   1:L PR[91] R[100]mm/sec CNT100;
   1:  PR[GP1:91,1] = PR[GP1:90,1] + 8.186;
   1:  PR[GP1:91,2] = PR[GP1:90,2] + 28.970;
   1:L PR[91] R[100]mm/sec CNT100;
   1:  PR[GP1:91,1] = PR[GP1:90,1] + 5.674;
   1:  PR[GP1:91,2] = PR[GP1:90,2] + 27.004;
   1:L PR[91] R[100]mm/sec CNT100;
   1:  PR[GP1:91,1] = PR[GP1:90,1] + 3.715;
   1:  PR[GP1:91,2] = PR[GP1:90,2] + 24.724;
   1:L PR[91] R[100]mm/sec CNT100;
   1:  PR[GP1:91,1] = PR[GP1:90,1] + 2.513;
   1:  PR[GP1:91,2] = PR[GP1:90,2] + 24.250;
   1:L PR[91] R[100]mm/sec CNT100;
   1:  PR[GP1:91,1] = PR[GP1:90,1] + 0.919;
   1:  PR[GP1:91,2] = PR[GP1:90,2] + 23.435;
   1:L PR[91] R[100]mm/sec CNT100;
   1:  ! -- Layer/Ebene 80 -- !;
   1:  PR[91] = PR[90];
   1:  PR[GP1:91,1] = PR[GP1:90,1] + -1.655;
   1:  PR[GP1:91,2] = PR[GP1:90,2] + 24.101;
   1:  PR[GP1:91,3] = PR[GP1:90,3] + 49.105;
   1:L PR[91] R[100]mm/sec CNT100;
   1:  PR[GP1:91,1] = PR[GP1:90,1] + -3.489;
   1:  PR[GP1:91,2] = PR[GP1:90,2] + 25.034;
   1:L PR[91] R[100]mm/sec CNT100;
   1:  PR[GP1:91,1] = PR[GP1:90,1] + -5.284;
   1:  PR[GP1:91,2] = PR[GP1:90,2] + 27.120;
   1:L PR[91] R[100]mm/sec CNT100;
   1:  PR[GP1:91,1] = PR[GP1:90,1] + -7.635;
   1:  PR[GP1:91,2] = PR[GP1:90,2] + 28.962;
   1:L PR[91] R[100]mm/sec CNT100;
   1:  PR[GP1:91,1] = PR[GP1:90,1] + -9.445;
   1:  PR[GP1:91,2] = PR[GP1:90,2] + 30.241;
   1:L PR[91] R[100]mm/sec CNT100;
   1:  PR[GP1:91,1] = PR[GP1:90,1] + -13.693;
   1:  PR[GP1:91,2] = PR[GP1:90,2] + 32.463;
   1:L PR[91] R[100]mm/sec CNT100;
   1:  PR[GP1:91,1] = PR[GP1:90,1] + -18.902;
   1:  PR[GP1:91,2] = PR[GP1:90,2] + 34.137;
   1:L PR[91] R[100]mm/sec CNT100;
   1:  PR[GP1:91,1] = PR[GP1:90,1] + -22.012;
   1:  PR[GP1:91,2] = PR[GP1:90,2] + 35.212;
   1:L PR[91] R[100]mm/sec CNT100;
   1:  PR[GP1:91,1] = PR[GP1:90,1] + -27.561;
   1:  PR[GP1:91,2] = PR[GP1:90,2] + 35.937;
   1:L PR[91] R[100]mm/sec CNT100;
   1:  PR[GP1:91,1] = PR[GP1:90,1] + -34.042;
   1:  PR[GP1:91,2] = PR[GP1:90,2] + 35.714;
   1:L PR[91] R[100]mm/sec CNT100;
   1:  PR[GP1:91,1] = PR[GP1:90,1] + -35.623;
   1:  PR[GP1:91,2] = PR[GP1:90,2] + 35.706;
   1:L PR[91] R[100]mm/sec CNT100;
   1:  PR[GP1:91,1] = PR[GP1:90,1] + -41.958;
   1:  PR[GP1:91,2] = PR[GP1:90,2] + 34.340;
   1:L PR[91] R[100]mm/sec CNT100;
   1:  PR[GP1:91,1] = PR[GP1:90,1] + -48.493;
   1:  PR[GP1:91,2] = PR[GP1:90,2] + 31.756;
   1:L PR[91] R[100]mm/sec CNT100;
   1:  PR[GP1:91,1] = PR[GP1:90,1] + -48.846;
   1:  PR[GP1:91,2] = PR[GP1:90,2] + 31.555;
   1:L PR[91] R[100]mm/sec CNT100;
   1:  PR[GP1:91,1] = PR[GP1:90,1] + -54.466;
   1:  PR[GP1:91,2] = PR[GP1:90,2] + 28.074;
   1:L PR[91] R[100]mm/sec CNT100;
   1:  PR[GP1:91,1] = PR[GP1:90,1] + -58.125;
   1:  PR[GP1:91,2] = PR[GP1:90,2] + 24.793;
   1:L PR[91] R[100]mm/sec CNT100;
   1:  PR[GP1:91,1] = PR[GP1:90,1] + -60.260;
   1:  PR[GP1:91,2] = PR[GP1:90,2] + 22.549;
   1:L PR[91] R[100]mm/sec CNT100;
   1:  PR[GP1:91,1] = PR[GP1:90,1] + -62.974;
   1:  PR[GP1:91,2] = PR[GP1:90,2] + 19.027;
   1:L PR[91] R[100]mm/sec CNT100;
   1:  PR[GP1:91,1] = PR[GP1:90,1] + -66.753;
   1:  PR[GP1:91,2] = PR[GP1:90,2] + 11.501;
   1:L PR[91] R[100]mm/sec CNT100;
   1:  PR[GP1:91,1] = PR[GP1:90,1] + -67.720;
   1:  PR[GP1:91,2] = PR[GP1:90,2] + 8.218;
   1:L PR[91] R[100]mm/sec CNT100;
   1:  PR[GP1:91,1] = PR[GP1:90,1] + -68.513;
   1:  PR[GP1:91,2] = PR[GP1:90,2] + 3.130;
   1:L PR[91] R[100]mm/sec CNT100;
   1:  PR[GP1:91,1] = PR[GP1:90,1] + -68.799;
   1:  PR[GP1:91,2] = PR[GP1:90,2] + -0.052;
   1:L PR[91] R[100]mm/sec CNT100;
   1:  PR[GP1:91,1] = PR[GP1:90,1] + -68.008;
   1:  PR[GP1:91,2] = PR[GP1:90,2] + -5.062;
   1:L PR[91] R[100]mm/sec CNT100;
   1:  PR[GP1:91,1] = PR[GP1:90,1] + -67.714;
   1:  PR[GP1:91,2] = PR[GP1:90,2] + -8.382;
   1:L PR[91] R[100]mm/sec CNT100;
   1:  PR[GP1:91,1] = PR[GP1:90,1] + -66.753;
   1:  PR[GP1:91,2] = PR[GP1:90,2] + -11.645;
   1:L PR[91] R[100]mm/sec CNT100;
   1:  PR[GP1:91,1] = PR[GP1:90,1] + -62.974;
   1:  PR[GP1:91,2] = PR[GP1:90,2] + -19.171;
   1:L PR[91] R[100]mm/sec CNT100;
   1:  PR[GP1:91,1] = PR[GP1:90,1] + -60.260;
   1:  PR[GP1:91,2] = PR[GP1:90,2] + -22.693;
   1:L PR[91] R[100]mm/sec CNT100;
   1:  PR[GP1:91,1] = PR[GP1:90,1] + -58.125;
   1:  PR[GP1:91,2] = PR[GP1:90,2] + -24.937;
   1:L PR[91] R[100]mm/sec CNT100;
   1:  PR[GP1:91,1] = PR[GP1:90,1] + -54.475;
   1:  PR[GP1:91,2] = PR[GP1:90,2] + -28.209;
   1:L PR[91] R[100]mm/sec CNT100;
   1:  PR[GP1:91,1] = PR[GP1:90,1] + -53.023;
   1:  PR[GP1:91,2] = PR[GP1:90,2] + -29.026;
   1:L PR[91] R[100]mm/sec CNT100;
   1:  PR[GP1:91,1] = PR[GP1:90,1] + -48.478;
   1:  PR[GP1:91,2] = PR[GP1:90,2] + -31.906;
   1:L PR[91] R[100]mm/sec CNT100;
   1:  PR[GP1:91,1] = PR[GP1:90,1] + -42.525;
   1:  PR[GP1:91,2] = PR[GP1:90,2] + -34.285;
   1:L PR[91] R[100]mm/sec CNT100;
   1:  PR[GP1:91,1] = PR[GP1:90,1] + -41.968;
   1:  PR[GP1:91,2] = PR[GP1:90,2] + -34.481;
   1:L PR[91] R[100]mm/sec CNT100;
   1:  PR[GP1:91,1] = PR[GP1:90,1] + -35.611;
   1:  PR[GP1:91,2] = PR[GP1:90,2] + -35.853;
   1:L PR[91] R[100]mm/sec CNT100;
   1:  PR[GP1:91,1] = PR[GP1:90,1] + -29.859;
   1:  PR[GP1:91,2] = PR[GP1:90,2] + -36.074;
   1:L PR[91] R[100]mm/sec CNT100;
   1:  PR[GP1:91,1] = PR[GP1:90,1] + -27.566;
   1:  PR[GP1:91,2] = PR[GP1:90,2] + -36.082;
   1:L PR[91] R[100]mm/sec CNT100;
   1:  PR[GP1:91,1] = PR[GP1:90,1] + -22.000;
   1:  PR[GP1:91,2] = PR[GP1:90,2] + -35.354;
   1:L PR[91] R[100]mm/sec CNT100;
   1:  PR[GP1:91,1] = PR[GP1:90,1] + -17.241;
   1:  PR[GP1:91,2] = PR[GP1:90,2] + -33.840;
   1:L PR[91] R[100]mm/sec CNT100;
   1:  PR[GP1:91,1] = PR[GP1:90,1] + -13.693;
   1:  PR[GP1:91,2] = PR[GP1:90,2] + -32.607;
   1:L PR[91] R[100]mm/sec CNT100;
   1:  PR[GP1:91,1] = PR[GP1:90,1] + -9.445;
   1:  PR[GP1:91,2] = PR[GP1:90,2] + -30.384;
   1:L PR[91] R[100]mm/sec CNT100;
   1:  PR[GP1:91,1] = PR[GP1:90,1] + -6.941;
   1:  PR[GP1:91,2] = PR[GP1:90,2] + -28.565;
   1:L PR[91] R[100]mm/sec CNT100;
   1:  PR[GP1:91,1] = PR[GP1:90,1] + -4.974;
   1:  PR[GP1:91,2] = PR[GP1:90,2] + -27.025;
   1:L PR[91] R[100]mm/sec CNT100;
   1:  PR[GP1:91,1] = PR[GP1:90,1] + -3.432;
   1:  PR[GP1:91,2] = PR[GP1:90,2] + -25.237;
   1:L PR[91] R[100]mm/sec CNT100;
   1:  PR[GP1:91,1] = PR[GP1:90,1] + -0.633;
   1:  PR[GP1:91,2] = PR[GP1:90,2] + -24.636;
   1:L PR[91] R[100]mm/sec CNT100;
   1:  PR[GP1:91,1] = PR[GP1:90,1] + 0.846;
   1:  PR[GP1:91,2] = PR[GP1:90,2] + -23.852;
   1:L PR[91] R[100]mm/sec CNT100;
   1:  PR[GP1:91,1] = PR[GP1:90,1] + 3.702;
   1:  PR[GP1:91,2] = PR[GP1:90,2] + -25.300;
   1:L PR[91] R[100]mm/sec CNT100;
   1:  PR[GP1:91,1] = PR[GP1:90,1] + 5.203;
   1:  PR[GP1:91,2] = PR[GP1:90,2] + -27.043;
   1:L PR[91] R[100]mm/sec CNT100;
   1:  PR[GP1:91,1] = PR[GP1:90,1] + 7.161;
   1:  PR[GP1:91,2] = PR[GP1:90,2] + -28.575;
   1:L PR[91] R[100]mm/sec CNT100;
   1:  PR[GP1:91,1] = PR[GP1:90,1] + 9.670;
   1:  PR[GP1:91,2] = PR[GP1:90,2] + -30.398;
   1:L PR[91] R[100]mm/sec CNT100;
   1:  PR[GP1:91,1] = PR[GP1:90,1] + 13.886;
   1:  PR[GP1:91,2] = PR[GP1:90,2] + -32.598;
   1:L PR[91] R[100]mm/sec CNT100;
   1:  PR[GP1:91,1] = PR[GP1:90,1] + 19.101;
   1:  PR[GP1:91,2] = PR[GP1:90,2] + -34.273;
   1:L PR[91] R[100]mm/sec CNT100;
   1:  PR[GP1:91,1] = PR[GP1:90,1] + 22.216;
   1:  PR[GP1:91,2] = PR[GP1:90,2] + -35.352;
   1:L PR[91] R[100]mm/sec CNT100;
   1:  PR[GP1:91,1] = PR[GP1:90,1] + 27.757;
   1:  PR[GP1:91,2] = PR[GP1:90,2] + -36.080;
   1:L PR[91] R[100]mm/sec CNT100;
   1:  PR[GP1:91,1] = PR[GP1:90,1] + 34.208;
   1:  PR[GP1:91,2] = PR[GP1:90,2] + -35.863;
   1:L PR[91] R[100]mm/sec CNT100;
   1:  PR[GP1:91,1] = PR[GP1:90,1] + 35.795;
   1:  PR[GP1:91,2] = PR[GP1:90,2] + -35.856;
   1:L PR[91] R[100]mm/sec CNT100;
   1:  PR[GP1:91,1] = PR[GP1:90,1] + 42.121;
   1:  PR[GP1:91,2] = PR[GP1:90,2] + -34.495;
   1:L PR[91] R[100]mm/sec CNT100;
   1:  PR[GP1:91,1] = PR[GP1:90,1] + 48.675;
   1:  PR[GP1:91,2] = PR[GP1:90,2] + -31.916;
   1:L PR[91] R[100]mm/sec CNT100;
   1:  PR[GP1:91,1] = PR[GP1:90,1] + 49.019;
   1:  PR[GP1:91,2] = PR[GP1:90,2] + -31.721;
   1:L PR[91] R[100]mm/sec CNT100;
   1:  PR[GP1:91,1] = PR[GP1:90,1] + 54.625;
   1:  PR[GP1:91,2] = PR[GP1:90,2] + -28.264;
   1:L PR[91] R[100]mm/sec CNT100;
   1:  PR[GP1:91,1] = PR[GP1:90,1] + 58.282;
   1:  PR[GP1:91,2] = PR[GP1:90,2] + -24.997;
   1:L PR[91] R[100]mm/sec CNT100;
   1:  PR[GP1:91,1] = PR[GP1:90,1] + 60.409;
   1:  PR[GP1:91,2] = PR[GP1:90,2] + -22.753;
   1:L PR[91] R[100]mm/sec CNT100;
   1:  PR[GP1:91,1] = PR[GP1:90,1] + 63.163;
   1:  PR[GP1:91,2] = PR[GP1:90,2] + -19.189;
   1:L PR[91] R[100]mm/sec CNT100;
   1:  PR[GP1:91,1] = PR[GP1:90,1] + 65.072;
   1:  PR[GP1:91,2] = PR[GP1:90,2] + -15.389;
   1:L PR[91] R[100]mm/sec CNT100;
   1:  PR[GP1:91,1] = PR[GP1:90,1] + 66.952;
   1:  PR[GP1:91,2] = PR[GP1:90,2] + -11.706;
   1:L PR[91] R[100]mm/sec CNT100;
   1:  PR[GP1:91,1] = PR[GP1:90,1] + 67.918;
   1:  PR[GP1:91,2] = PR[GP1:90,2] + -8.468;
   1:L PR[91] R[100]mm/sec CNT100;
   1:  PR[GP1:91,1] = PR[GP1:90,1] + 68.711;
   1:  PR[GP1:91,2] = PR[GP1:90,2] + -3.366;
   1:L PR[91] R[100]mm/sec CNT100;
   1:  PR[GP1:91,1] = PR[GP1:90,1] + 69.012;
   1:  PR[GP1:91,2] = PR[GP1:90,2] + -0.092;
   1:L PR[91] R[100]mm/sec CNT100;
   1:  PR[GP1:91,1] = PR[GP1:90,1] + 68.221;
   1:  PR[GP1:91,2] = PR[GP1:90,2] + 4.931;
   1:L PR[91] R[100]mm/sec CNT100;
   1:  PR[GP1:91,1] = PR[GP1:90,1] + 67.912;
   1:  PR[GP1:91,2] = PR[GP1:90,2] + 8.343;
   1:L PR[91] R[100]mm/sec CNT100;
   1:  PR[GP1:91,1] = PR[GP1:90,1] + 66.951;
   1:  PR[GP1:91,2] = PR[GP1:90,2] + 11.564;
   1:L PR[91] R[100]mm/sec CNT100;
   1:  PR[GP1:91,1] = PR[GP1:90,1] + 64.946;
   1:  PR[GP1:91,2] = PR[GP1:90,2] + 15.559;
   1:L PR[91] R[100]mm/sec CNT100;
   1:  PR[GP1:91,1] = PR[GP1:90,1] + 63.164;
   1:  PR[GP1:91,2] = PR[GP1:90,2] + 19.044;
   1:L PR[91] R[100]mm/sec CNT100;
   1:  PR[GP1:91,1] = PR[GP1:90,1] + 60.409;
   1:  PR[GP1:91,2] = PR[GP1:90,2] + 22.609;
   1:L PR[91] R[100]mm/sec CNT100;
   1:  PR[GP1:91,1] = PR[GP1:90,1] + 58.282;
   1:  PR[GP1:91,2] = PR[GP1:90,2] + 24.853;
   1:L PR[91] R[100]mm/sec CNT100;
   1:  PR[GP1:91,1] = PR[GP1:90,1] + 54.634;
   1:  PR[GP1:91,2] = PR[GP1:90,2] + 28.112;
   1:L PR[91] R[100]mm/sec CNT100;
   1:  PR[GP1:91,1] = PR[GP1:90,1] + 53.192;
   1:  PR[GP1:91,2] = PR[GP1:90,2] + 28.923;
   1:L PR[91] R[100]mm/sec CNT100;
   1:  PR[GP1:91,1] = PR[GP1:90,1] + 48.661;
   1:  PR[GP1:91,2] = PR[GP1:90,2] + 31.778;
   1:L PR[91] R[100]mm/sec CNT100;
   1:  PR[GP1:91,1] = PR[GP1:90,1] + 42.696;
   1:  PR[GP1:91,2] = PR[GP1:90,2] + 34.150;
   1:L PR[91] R[100]mm/sec CNT100;
   1:  PR[GP1:91,1] = PR[GP1:90,1] + 42.133;
   1:  PR[GP1:91,2] = PR[GP1:90,2] + 34.349;
   1:L PR[91] R[100]mm/sec CNT100;
   1:  PR[GP1:91,1] = PR[GP1:90,1] + 35.787;
   1:  PR[GP1:91,2] = PR[GP1:90,2] + 35.714;
   1:L PR[91] R[100]mm/sec CNT100;
   1:  PR[GP1:91,1] = PR[GP1:90,1] + 30.063;
   1:  PR[GP1:91,2] = PR[GP1:90,2] + 35.930;
   1:L PR[91] R[100]mm/sec CNT100;
   1:  PR[GP1:91,1] = PR[GP1:90,1] + 27.770;
   1:  PR[GP1:91,2] = PR[GP1:90,2] + 35.938;
   1:L PR[91] R[100]mm/sec CNT100;
   1:  PR[GP1:91,1] = PR[GP1:90,1] + 22.213;
   1:  PR[GP1:91,2] = PR[GP1:90,2] + 35.208;
   1:L PR[91] R[100]mm/sec CNT100;
   1:  PR[GP1:91,1] = PR[GP1:90,1] + 17.448;
   1:  PR[GP1:91,2] = PR[GP1:90,2] + 33.692;
   1:L PR[91] R[100]mm/sec CNT100;
   1:  PR[GP1:91,1] = PR[GP1:90,1] + 13.898;
   1:  PR[GP1:91,2] = PR[GP1:90,2] + 32.461;
   1:L PR[91] R[100]mm/sec CNT100;
   1:  PR[GP1:91,1] = PR[GP1:90,1] + 9.670;
   1:  PR[GP1:91,2] = PR[GP1:90,2] + 30.255;
   1:L PR[91] R[100]mm/sec CNT100;
   1:  PR[GP1:91,1] = PR[GP1:90,1] + 7.856;
   1:  PR[GP1:91,2] = PR[GP1:90,2] + 28.973;
   1:L PR[91] R[100]mm/sec CNT100;
   1:  PR[GP1:91,1] = PR[GP1:90,1] + 5.516;
   1:  PR[GP1:91,2] = PR[GP1:90,2] + 27.142;
   1:L PR[91] R[100]mm/sec CNT100;
   1:  PR[GP1:91,1] = PR[GP1:90,1] + 3.685;
   1:  PR[GP1:91,2] = PR[GP1:90,2] + 25.011;
   1:L PR[91] R[100]mm/sec CNT100;
   1:  PR[GP1:91,1] = PR[GP1:90,1] + 2.424;
   1:  PR[GP1:91,2] = PR[GP1:90,2] + 24.513;
   1:L PR[91] R[100]mm/sec CNT100;
   1:  PR[GP1:91,1] = PR[GP1:90,1] + 0.960;
   1:  PR[GP1:91,2] = PR[GP1:90,2] + 23.765;
   1:L PR[91] R[100]mm/sec CNT100;
   1:  ! -- Layer/Ebene 81 -- !;
   1:  PR[91] = PR[90];
   1:  PR[GP1:91,1] = PR[GP1:90,1] + -1.744;
   1:  PR[GP1:91,2] = PR[GP1:90,2] + 24.447;
   1:  PR[GP1:91,3] = PR[GP1:90,3] + 49.715;
   1:L PR[91] R[100]mm/sec CNT100;
   1:  PR[GP1:91,1] = PR[GP1:90,1] + -3.460;
   1:  PR[GP1:91,2] = PR[GP1:90,2] + 25.320;
   1:L PR[91] R[100]mm/sec CNT100;
   1:  PR[GP1:91,1] = PR[GP1:90,1] + -5.128;
   1:  PR[GP1:91,2] = PR[GP1:90,2] + 27.260;
   1:L PR[91] R[100]mm/sec CNT100;
   1:  PR[GP1:91,1] = PR[GP1:90,1] + -7.305;
   1:  PR[GP1:91,2] = PR[GP1:90,2] + 28.965;
   1:L PR[91] R[100]mm/sec CNT100;
   1:  PR[GP1:91,1] = PR[GP1:90,1] + -9.235;
   1:  PR[GP1:91,2] = PR[GP1:90,2] + 30.328;
   1:L PR[91] R[100]mm/sec CNT100;
   1:  PR[GP1:91,1] = PR[GP1:90,1] + -13.351;
   1:  PR[GP1:91,2] = PR[GP1:90,2] + 32.482;
   1:L PR[91] R[100]mm/sec CNT100;
   1:  PR[GP1:91,1] = PR[GP1:90,1] + -18.401;
   1:  PR[GP1:91,2] = PR[GP1:90,2] + 34.104;
   1:L PR[91] R[100]mm/sec CNT100;
   1:  PR[GP1:91,1] = PR[GP1:90,1] + -21.813;
   1:  PR[GP1:91,2] = PR[GP1:90,2] + 35.284;
   1:L PR[91] R[100]mm/sec CNT100;
   1:  PR[GP1:91,1] = PR[GP1:90,1] + -27.209;
   1:  PR[GP1:91,2] = PR[GP1:90,2] + 35.989;
   1:L PR[91] R[100]mm/sec CNT100;
   1:  PR[GP1:91,1] = PR[GP1:90,1] + -33.514;
   1:  PR[GP1:91,2] = PR[GP1:90,2] + 35.773;
   1:L PR[91] R[100]mm/sec CNT100;
   1:  PR[GP1:91,1] = PR[GP1:90,1] + -35.435;
   1:  PR[GP1:91,2] = PR[GP1:90,2] + 35.763;
   1:L PR[91] R[100]mm/sec CNT100;
   1:  PR[GP1:91,1] = PR[GP1:90,1] + -41.613;
   1:  PR[GP1:91,2] = PR[GP1:90,2] + 34.430;
   1:L PR[91] R[100]mm/sec CNT100;
   1:  PR[GP1:91,1] = PR[GP1:90,1] + -48.418;
   1:  PR[GP1:91,2] = PR[GP1:90,2] + 31.741;
   1:L PR[91] R[100]mm/sec CNT100;
   1:  PR[GP1:91,1] = PR[GP1:90,1] + -54.253;
   1:  PR[GP1:91,2] = PR[GP1:90,2] + 28.124;
   1:L PR[91] R[100]mm/sec CNT100;
   1:  PR[GP1:91,1] = PR[GP1:90,1] + -58.181;
   1:  PR[GP1:91,2] = PR[GP1:90,2] + 24.602;
   1:L PR[91] R[100]mm/sec CNT100;
   1:  PR[GP1:91,1] = PR[GP1:90,1] + -59.893;
   1:  PR[GP1:91,2] = PR[GP1:90,2] + 22.802;
   1:L PR[91] R[100]mm/sec CNT100;
   1:  PR[GP1:91,1] = PR[GP1:90,1] + -62.849;
   1:  PR[GP1:91,2] = PR[GP1:90,2] + 18.966;
   1:L PR[91] R[100]mm/sec CNT100;
   1:  PR[GP1:91,1] = PR[GP1:90,1] + -66.536;
   1:  PR[GP1:91,2] = PR[GP1:90,2] + 11.628;
   1:L PR[91] R[100]mm/sec CNT100;
   1:  PR[GP1:91,1] = PR[GP1:90,1] + -67.603;
   1:  PR[GP1:91,2] = PR[GP1:90,2] + 8.004;
   1:L PR[91] R[100]mm/sec CNT100;
   1:  PR[GP1:91,1] = PR[GP1:90,1] + -68.306;
   1:  PR[GP1:91,2] = PR[GP1:90,2] + 3.493;
   1:L PR[91] R[100]mm/sec CNT100;
   1:  PR[GP1:91,1] = PR[GP1:90,1] + -68.625;
   1:  PR[GP1:91,2] = PR[GP1:90,2] + -0.052;
   1:L PR[91] R[100]mm/sec CNT100;
   1:  PR[GP1:91,1] = PR[GP1:90,1] + -67.921;
   1:  PR[GP1:91,2] = PR[GP1:90,2] + -4.508;
   1:L PR[91] R[100]mm/sec CNT100;
   1:  PR[GP1:91,1] = PR[GP1:90,1] + -67.597;
   1:  PR[GP1:91,2] = PR[GP1:90,2] + -8.168;
   1:L PR[91] R[100]mm/sec CNT100;
   1:  PR[GP1:91,1] = PR[GP1:90,1] + -66.536;
   1:  PR[GP1:91,2] = PR[GP1:90,2] + -11.772;
   1:L PR[91] R[100]mm/sec CNT100;
   1:  PR[GP1:91,1] = PR[GP1:90,1] + -62.849;
   1:  PR[GP1:91,2] = PR[GP1:90,2] + -19.110;
   1:L PR[91] R[100]mm/sec CNT100;
   1:  PR[GP1:91,1] = PR[GP1:90,1] + -59.893;
   1:  PR[GP1:91,2] = PR[GP1:90,2] + -22.946;
   1:L PR[91] R[100]mm/sec CNT100;
   1:  PR[GP1:91,1] = PR[GP1:90,1] + -58.181;
   1:  PR[GP1:91,2] = PR[GP1:90,2] + -24.746;
   1:L PR[91] R[100]mm/sec CNT100;
   1:  PR[GP1:91,1] = PR[GP1:90,1] + -54.262;
   1:  PR[GP1:91,2] = PR[GP1:90,2] + -28.259;
   1:L PR[91] R[100]mm/sec CNT100;
   1:  PR[GP1:91,1] = PR[GP1:90,1] + -53.300;
   1:  PR[GP1:91,2] = PR[GP1:90,2] + -28.801;
   1:L PR[91] R[100]mm/sec CNT100;
   1:  PR[GP1:91,1] = PR[GP1:90,1] + -48.414;
   1:  PR[GP1:91,2] = PR[GP1:90,2] + -31.887;
   1:L PR[91] R[100]mm/sec CNT100;
   1:  PR[GP1:91,1] = PR[GP1:90,1] + -42.479;
   1:  PR[GP1:91,2] = PR[GP1:90,2] + -34.270;
   1:L PR[91] R[100]mm/sec CNT100;
   1:  PR[GP1:91,1] = PR[GP1:90,1] + -41.622;
   1:  PR[GP1:91,2] = PR[GP1:90,2] + -34.572;
   1:L PR[91] R[100]mm/sec CNT100;
   1:  PR[GP1:91,1] = PR[GP1:90,1] + -35.423;
   1:  PR[GP1:91,2] = PR[GP1:90,2] + -35.909;
   1:L PR[91] R[100]mm/sec CNT100;
   1:  PR[GP1:91,1] = PR[GP1:90,1] + -29.813;
   1:  PR[GP1:91,2] = PR[GP1:90,2] + -36.126;
   1:L PR[91] R[100]mm/sec CNT100;
   1:  PR[GP1:91,1] = PR[GP1:90,1] + -27.214;
   1:  PR[GP1:91,2] = PR[GP1:90,2] + -36.134;
   1:L PR[91] R[100]mm/sec CNT100;
   1:  PR[GP1:91,1] = PR[GP1:90,1] + -21.801;
   1:  PR[GP1:91,2] = PR[GP1:90,2] + -35.426;
   1:L PR[91] R[100]mm/sec CNT100;
   1:  PR[GP1:91,1] = PR[GP1:90,1] + -17.172;
   1:  PR[GP1:91,2] = PR[GP1:90,2] + -33.953;
   1:L PR[91] R[100]mm/sec CNT100;
   1:  PR[GP1:91,1] = PR[GP1:90,1] + -13.351;
   1:  PR[GP1:91,2] = PR[GP1:90,2] + -32.625;
   1:L PR[91] R[100]mm/sec CNT100;
   1:  PR[GP1:91,1] = PR[GP1:90,1] + -9.234;
   1:  PR[GP1:91,2] = PR[GP1:90,2] + -30.472;
   1:L PR[91] R[100]mm/sec CNT100;
   1:  PR[GP1:91,1] = PR[GP1:90,1] + -6.567;
   1:  PR[GP1:91,2] = PR[GP1:90,2] + -28.534;
   1:L PR[91] R[100]mm/sec CNT100;
   1:  PR[GP1:91,1] = PR[GP1:90,1] + -4.801;
   1:  PR[GP1:91,2] = PR[GP1:90,2] + -27.151;
   1:L PR[91] R[100]mm/sec CNT100;
   1:  PR[GP1:91,1] = PR[GP1:90,1] + -3.403;
   1:  PR[GP1:91,2] = PR[GP1:90,2] + -25.530;
   1:L PR[91] R[100]mm/sec CNT100;
   1:  PR[GP1:91,1] = PR[GP1:90,1] + -0.466;
   1:  PR[GP1:91,2] = PR[GP1:90,2] + -24.899;
   1:L PR[91] R[100]mm/sec CNT100;
   1:  PR[GP1:91,1] = PR[GP1:90,1] + 0.887;
   1:  PR[GP1:91,2] = PR[GP1:90,2] + -24.182;
   1:L PR[91] R[100]mm/sec CNT100;
   1:  PR[GP1:91,1] = PR[GP1:90,1] + 3.672;
   1:  PR[GP1:91,2] = PR[GP1:90,2] + -25.593;
   1:L PR[91] R[100]mm/sec CNT100;
   1:  PR[GP1:91,1] = PR[GP1:90,1] + 5.028;
   1:  PR[GP1:91,2] = PR[GP1:90,2] + -27.168;
   1:L PR[91] R[100]mm/sec CNT100;
   1:  PR[GP1:91,1] = PR[GP1:90,1] + 6.786;
   1:  PR[GP1:91,2] = PR[GP1:90,2] + -28.543;
   1:L PR[91] R[100]mm/sec CNT100;
   1:  PR[GP1:91,1] = PR[GP1:90,1] + 9.459;
   1:  PR[GP1:91,2] = PR[GP1:90,2] + -30.485;
   1:L PR[91] R[100]mm/sec CNT100;
   1:  PR[GP1:91,1] = PR[GP1:90,1] + 13.544;
   1:  PR[GP1:91,2] = PR[GP1:90,2] + -32.617;
   1:L PR[91] R[100]mm/sec CNT100;
   1:  PR[GP1:91,1] = PR[GP1:90,1] + 18.599;
   1:  PR[GP1:91,2] = PR[GP1:90,2] + -34.241;
   1:L PR[91] R[100]mm/sec CNT100;
   1:  PR[GP1:91,1] = PR[GP1:90,1] + 22.017;
   1:  PR[GP1:91,2] = PR[GP1:90,2] + -35.424;
   1:L PR[91] R[100]mm/sec CNT100;
   1:  PR[GP1:91,1] = PR[GP1:90,1] + 27.405;
   1:  PR[GP1:91,2] = PR[GP1:90,2] + -36.133;
   1:L PR[91] R[100]mm/sec CNT100;
   1:  PR[GP1:91,1] = PR[GP1:90,1] + 33.681;
   1:  PR[GP1:91,2] = PR[GP1:90,2] + -35.921;
   1:L PR[91] R[100]mm/sec CNT100;
   1:  PR[GP1:91,1] = PR[GP1:90,1] + 35.608;
   1:  PR[GP1:91,2] = PR[GP1:90,2] + -35.913;
   1:L PR[91] R[100]mm/sec CNT100;
   1:  PR[GP1:91,1] = PR[GP1:90,1] + 41.777;
   1:  PR[GP1:91,2] = PR[GP1:90,2] + -34.585;
   1:L PR[91] R[100]mm/sec CNT100;
   1:  PR[GP1:91,1] = PR[GP1:90,1] + 48.597;
   1:  PR[GP1:91,2] = PR[GP1:90,2] + -31.903;
   1:L PR[91] R[100]mm/sec CNT100;
   1:  PR[GP1:91,1] = PR[GP1:90,1] + 54.408;
   1:  PR[GP1:91,2] = PR[GP1:90,2] + -28.317;
   1:L PR[91] R[100]mm/sec CNT100;
   1:  PR[GP1:91,1] = PR[GP1:90,1] + 58.334;
   1:  PR[GP1:91,2] = PR[GP1:90,2] + -24.809;
   1:L PR[91] R[100]mm/sec CNT100;
   1:  PR[GP1:91,1] = PR[GP1:90,1] + 60.037;
   1:  PR[GP1:91,2] = PR[GP1:90,2] + -23.013;
   1:L PR[91] R[100]mm/sec CNT100;
   1:  PR[GP1:91,1] = PR[GP1:90,1] + 63.036;
   1:  PR[GP1:91,2] = PR[GP1:90,2] + -19.131;
   1:L PR[91] R[100]mm/sec CNT100;
   1:  PR[GP1:91,1] = PR[GP1:90,1] + 64.662;
   1:  PR[GP1:91,2] = PR[GP1:90,2] + -15.896;
   1:L PR[91] R[100]mm/sec CNT100;
   1:  PR[GP1:91,1] = PR[GP1:90,1] + 66.733;
   1:  PR[GP1:91,2] = PR[GP1:90,2] + -11.836;
   1:L PR[91] R[100]mm/sec CNT100;
   1:  PR[GP1:91,1] = PR[GP1:90,1] + 67.800;
   1:  PR[GP1:91,2] = PR[GP1:90,2] + -8.262;
   1:L PR[91] R[100]mm/sec CNT100;
   1:  PR[GP1:91,1] = PR[GP1:90,1] + 68.503;
   1:  PR[GP1:91,2] = PR[GP1:90,2] + -3.740;
   1:L PR[91] R[100]mm/sec CNT100;
   1:  PR[GP1:91,1] = PR[GP1:90,1] + 68.838;
   1:  PR[GP1:91,2] = PR[GP1:90,2] + -0.092;
   1:L PR[91] R[100]mm/sec CNT100;
   1:  PR[GP1:91,1] = PR[GP1:90,1] + 68.134;
   1:  PR[GP1:91,2] = PR[GP1:90,2] + 4.377;
   1:L PR[91] R[100]mm/sec CNT100;
   1:  PR[GP1:91,1] = PR[GP1:90,1] + 67.794;
   1:  PR[GP1:91,2] = PR[GP1:90,2] + 8.137;
   1:L PR[91] R[100]mm/sec CNT100;
   1:  PR[GP1:91,1] = PR[GP1:90,1] + 66.733;
   1:  PR[GP1:91,2] = PR[GP1:90,2] + 11.694;
   1:L PR[91] R[100]mm/sec CNT100;
   1:  PR[GP1:91,1] = PR[GP1:90,1] + 64.977;
   1:  PR[GP1:91,2] = PR[GP1:90,2] + 15.191;
   1:L PR[91] R[100]mm/sec CNT100;
   1:  PR[GP1:91,1] = PR[GP1:90,1] + 63.037;
   1:  PR[GP1:91,2] = PR[GP1:90,2] + 18.986;
   1:L PR[91] R[100]mm/sec CNT100;
   1:  PR[GP1:91,1] = PR[GP1:90,1] + 60.037;
   1:  PR[GP1:91,2] = PR[GP1:90,2] + 22.869;
   1:L PR[91] R[100]mm/sec CNT100;
   1:  PR[GP1:91,1] = PR[GP1:90,1] + 58.334;
   1:  PR[GP1:91,2] = PR[GP1:90,2] + 24.665;
   1:L PR[91] R[100]mm/sec CNT100;
   1:  PR[GP1:91,1] = PR[GP1:90,1] + 54.417;
   1:  PR[GP1:91,2] = PR[GP1:90,2] + 28.165;
   1:L PR[91] R[100]mm/sec CNT100;
   1:  PR[GP1:91,1] = PR[GP1:90,1] + 53.466;
   1:  PR[GP1:91,2] = PR[GP1:90,2] + 28.700;
   1:L PR[91] R[100]mm/sec CNT100;
   1:  PR[GP1:91,1] = PR[GP1:90,1] + 48.593;
   1:  PR[GP1:91,2] = PR[GP1:90,2] + 31.761;
   1:L PR[91] R[100]mm/sec CNT100;
   1:  PR[GP1:91,1] = PR[GP1:90,1] + 42.650;
   1:  PR[GP1:91,2] = PR[GP1:90,2] + 34.135;
   1:L PR[91] R[100]mm/sec CNT100;
   1:  PR[GP1:91,1] = PR[GP1:90,1] + 41.788;
   1:  PR[GP1:91,2] = PR[GP1:90,2] + 34.439;
   1:L PR[91] R[100]mm/sec CNT100;
   1:  PR[GP1:91,1] = PR[GP1:90,1] + 35.600;
   1:  PR[GP1:91,2] = PR[GP1:90,2] + 35.771;
   1:L PR[91] R[100]mm/sec CNT100;
   1:  PR[GP1:91,1] = PR[GP1:90,1] + 30.018;
   1:  PR[GP1:91,2] = PR[GP1:90,2] + 35.981;
   1:L PR[91] R[100]mm/sec CNT100;
   1:  PR[GP1:91,1] = PR[GP1:90,1] + 27.419;
   1:  PR[GP1:91,2] = PR[GP1:90,2] + 35.990;
   1:L PR[91] R[100]mm/sec CNT100;
   1:  PR[GP1:91,1] = PR[GP1:90,1] + 22.014;
   1:  PR[GP1:91,2] = PR[GP1:90,2] + 35.280;
   1:L PR[91] R[100]mm/sec CNT100;
   1:  PR[GP1:91,1] = PR[GP1:90,1] + 17.380;
   1:  PR[GP1:91,2] = PR[GP1:90,2] + 33.805;
   1:L PR[91] R[100]mm/sec CNT100;
   1:  PR[GP1:91,1] = PR[GP1:90,1] + 13.556;
   1:  PR[GP1:91,2] = PR[GP1:90,2] + 32.480;
   1:L PR[91] R[100]mm/sec CNT100;
   1:  PR[GP1:91,1] = PR[GP1:90,1] + 9.459;
   1:  PR[GP1:91,2] = PR[GP1:90,2] + 30.341;
   1:L PR[91] R[100]mm/sec CNT100;
   1:  PR[GP1:91,1] = PR[GP1:90,1] + 7.525;
   1:  PR[GP1:91,2] = PR[GP1:90,2] + 28.975;
   1:L PR[91] R[100]mm/sec CNT100;
   1:  PR[GP1:91,1] = PR[GP1:90,1] + 5.358;
   1:  PR[GP1:91,2] = PR[GP1:90,2] + 27.280;
   1:L PR[91] R[100]mm/sec CNT100;
   1:  PR[GP1:91,1] = PR[GP1:90,1] + 3.655;
   1:  PR[GP1:91,2] = PR[GP1:90,2] + 25.298;
   1:L PR[91] R[100]mm/sec CNT100;
   1:  PR[GP1:91,1] = PR[GP1:90,1] + 2.335;
   1:  PR[GP1:91,2] = PR[GP1:90,2] + 24.776;
   1:L PR[91] R[100]mm/sec CNT100;
   1:  PR[GP1:91,1] = PR[GP1:90,1] + 1.001;
   1:  PR[GP1:91,2] = PR[GP1:90,2] + 24.095;
   1:L PR[91] R[100]mm/sec CNT100;
   1:  ! -- Layer/Ebene 82 -- !;
   1:  PR[91] = PR[90];
   1:  PR[GP1:91,1] = PR[GP1:90,1] + -1.832;
   1:  PR[GP1:91,2] = PR[GP1:90,2] + 24.794;
   1:  PR[GP1:91,3] = PR[GP1:90,3] + 50.325;
   1:L PR[91] R[100]mm/sec CNT100;
   1:  PR[GP1:91,1] = PR[GP1:90,1] + -3.430;
   1:  PR[GP1:91,2] = PR[GP1:90,2] + 25.607;
   1:L PR[91] R[100]mm/sec CNT100;
   1:  PR[GP1:91,1] = PR[GP1:90,1] + -4.972;
   1:  PR[GP1:91,2] = PR[GP1:90,2] + 27.399;
   1:L PR[91] R[100]mm/sec CNT100;
   1:  PR[GP1:91,1] = PR[GP1:90,1] + -6.976;
   1:  PR[GP1:91,2] = PR[GP1:90,2] + 28.969;
   1:L PR[91] R[100]mm/sec CNT100;
   1:  PR[GP1:91,1] = PR[GP1:90,1] + -9.024;
   1:  PR[GP1:91,2] = PR[GP1:90,2] + 30.416;
   1:L PR[91] R[100]mm/sec CNT100;
   1:  PR[GP1:91,1] = PR[GP1:90,1] + -13.009;
   1:  PR[GP1:91,2] = PR[GP1:90,2] + 32.501;
   1:L PR[91] R[100]mm/sec CNT100;
   1:  PR[GP1:91,1] = PR[GP1:90,1] + -17.900;
   1:  PR[GP1:91,2] = PR[GP1:90,2] + 34.072;
   1:L PR[91] R[100]mm/sec CNT100;
   1:  PR[GP1:91,1] = PR[GP1:90,1] + -21.615;
   1:  PR[GP1:91,2] = PR[GP1:90,2] + 35.356;
   1:L PR[91] R[100]mm/sec CNT100;
   1:  PR[GP1:91,1] = PR[GP1:90,1] + -26.858;
   1:  PR[GP1:91,2] = PR[GP1:90,2] + 36.042;
   1:L PR[91] R[100]mm/sec CNT100;
   1:  PR[GP1:91,1] = PR[GP1:90,1] + -32.986;
   1:  PR[GP1:91,2] = PR[GP1:90,2] + 35.831;
   1:L PR[91] R[100]mm/sec CNT100;
   1:  PR[GP1:91,1] = PR[GP1:90,1] + -35.247;
   1:  PR[GP1:91,2] = PR[GP1:90,2] + 35.820;
   1:L PR[91] R[100]mm/sec CNT100;
   1:  PR[GP1:91,1] = PR[GP1:90,1] + -41.267;
   1:  PR[GP1:91,2] = PR[GP1:90,2] + 34.521;
   1:L PR[91] R[100]mm/sec CNT100;
   1:  PR[GP1:91,1] = PR[GP1:90,1] + -47.841;
   1:  PR[GP1:91,2] = PR[GP1:90,2] + 31.918;
   1:L PR[91] R[100]mm/sec CNT100;
   1:  PR[GP1:91,1] = PR[GP1:90,1] + -48.243;
   1:  PR[GP1:91,2] = PR[GP1:90,2] + 31.775;
   1:L PR[91] R[100]mm/sec CNT100;
   1:  PR[GP1:91,1] = PR[GP1:90,1] + -54.039;
   1:  PR[GP1:91,2] = PR[GP1:90,2] + 28.174;
   1:L PR[91] R[100]mm/sec CNT100;
   1:  PR[GP1:91,1] = PR[GP1:90,1] + -58.237;
   1:  PR[GP1:91,2] = PR[GP1:90,2] + 24.411;
   1:L PR[91] R[100]mm/sec CNT100;
   1:  PR[GP1:91,1] = PR[GP1:90,1] + -59.526;
   1:  PR[GP1:91,2] = PR[GP1:90,2] + 23.055;
   1:L PR[91] R[100]mm/sec CNT100;
   1:  PR[GP1:91,1] = PR[GP1:90,1] + -62.724;
   1:  PR[GP1:91,2] = PR[GP1:90,2] + 18.904;
   1:L PR[91] R[100]mm/sec CNT100;
   1:  PR[GP1:91,1] = PR[GP1:90,1] + -66.320;
   1:  PR[GP1:91,2] = PR[GP1:90,2] + 11.754;
   1:L PR[91] R[100]mm/sec CNT100;
   1:  PR[GP1:91,1] = PR[GP1:90,1] + -67.486;
   1:  PR[GP1:91,2] = PR[GP1:90,2] + 7.790;
   1:L PR[91] R[100]mm/sec CNT100;
   1:  PR[GP1:91,1] = PR[GP1:90,1] + -68.100;
   1:  PR[GP1:91,2] = PR[GP1:90,2] + 3.857;
   1:L PR[91] R[100]mm/sec CNT100;
   1:  PR[GP1:91,1] = PR[GP1:90,1] + -68.451;
   1:  PR[GP1:91,2] = PR[GP1:90,2] + -0.052;
   1:L PR[91] R[100]mm/sec CNT100;
   1:  PR[GP1:91,1] = PR[GP1:90,1] + -67.834;
   1:  PR[GP1:91,2] = PR[GP1:90,2] + -3.955;
   1:L PR[91] R[100]mm/sec CNT100;
   1:  PR[GP1:91,1] = PR[GP1:90,1] + -67.481;
   1:  PR[GP1:91,2] = PR[GP1:90,2] + -7.953;
   1:L PR[91] R[100]mm/sec CNT100;
   1:  PR[GP1:91,1] = PR[GP1:90,1] + -66.320;
   1:  PR[GP1:91,2] = PR[GP1:90,2] + -11.898;
   1:L PR[91] R[100]mm/sec CNT100;
   1:  PR[GP1:91,1] = PR[GP1:90,1] + -62.724;
   1:  PR[GP1:91,2] = PR[GP1:90,2] + -19.048;
   1:L PR[91] R[100]mm/sec CNT100;
   1:  PR[GP1:91,1] = PR[GP1:90,1] + -59.526;
   1:  PR[GP1:91,2] = PR[GP1:90,2] + -23.199;
   1:L PR[91] R[100]mm/sec CNT100;
   1:  PR[GP1:91,1] = PR[GP1:90,1] + -58.237;
   1:  PR[GP1:91,2] = PR[GP1:90,2] + -24.555;
   1:L PR[91] R[100]mm/sec CNT100;
   1:  PR[GP1:91,1] = PR[GP1:90,1] + -54.049;
   1:  PR[GP1:91,2] = PR[GP1:90,2] + -28.309;
   1:L PR[91] R[100]mm/sec CNT100;
   1:  PR[GP1:91,1] = PR[GP1:90,1] + -53.575;
   1:  PR[GP1:91,2] = PR[GP1:90,2] + -28.575;
   1:L PR[91] R[100]mm/sec CNT100;
   1:  PR[GP1:91,1] = PR[GP1:90,1] + -51.489;
   1:  PR[GP1:91,2] = PR[GP1:90,2] + -29.897;
   1:L PR[91] R[100]mm/sec CNT100;
   1:  PR[GP1:91,1] = PR[GP1:90,1] + -48.232;
   1:  PR[GP1:91,2] = PR[GP1:90,2] + -31.926;
   1:L PR[91] R[100]mm/sec CNT100;
   1:  PR[GP1:91,1] = PR[GP1:90,1] + -42.433;
   1:  PR[GP1:91,2] = PR[GP1:90,2] + -34.255;
   1:L PR[91] R[100]mm/sec CNT100;
   1:  PR[GP1:91,1] = PR[GP1:90,1] + -41.276;
   1:  PR[GP1:91,2] = PR[GP1:90,2] + -34.663;
   1:L PR[91] R[100]mm/sec CNT100;
   1:  PR[GP1:91,1] = PR[GP1:90,1] + -35.235;
   1:  PR[GP1:91,2] = PR[GP1:90,2] + -35.966;
   1:L PR[91] R[100]mm/sec CNT100;
   1:  PR[GP1:91,1] = PR[GP1:90,1] + -29.767;
   1:  PR[GP1:91,2] = PR[GP1:90,2] + -36.177;
   1:L PR[91] R[100]mm/sec CNT100;
   1:  PR[GP1:91,1] = PR[GP1:90,1] + -26.862;
   1:  PR[GP1:91,2] = PR[GP1:90,2] + -36.186;
   1:L PR[91] R[100]mm/sec CNT100;
   1:  PR[GP1:91,1] = PR[GP1:90,1] + -21.602;
   1:  PR[GP1:91,2] = PR[GP1:90,2] + -35.498;
   1:L PR[91] R[100]mm/sec CNT100;
   1:  PR[GP1:91,1] = PR[GP1:90,1] + -17.104;
   1:  PR[GP1:91,2] = PR[GP1:90,2] + -34.067;
   1:L PR[91] R[100]mm/sec CNT100;
   1:  PR[GP1:91,1] = PR[GP1:90,1] + -13.009;
   1:  PR[GP1:91,2] = PR[GP1:90,2] + -32.644;
   1:L PR[91] R[100]mm/sec CNT100;
   1:  PR[GP1:91,1] = PR[GP1:90,1] + -9.023;
   1:  PR[GP1:91,2] = PR[GP1:90,2] + -30.559;
   1:L PR[91] R[100]mm/sec CNT100;
   1:  PR[GP1:91,1] = PR[GP1:90,1] + -6.193;
   1:  PR[GP1:91,2] = PR[GP1:90,2] + -28.503;
   1:L PR[91] R[100]mm/sec CNT100;
   1:  PR[GP1:91,1] = PR[GP1:90,1] + -4.627;
   1:  PR[GP1:91,2] = PR[GP1:90,2] + -27.277;
   1:L PR[91] R[100]mm/sec CNT100;
   1:  PR[GP1:91,1] = PR[GP1:90,1] + -3.374;
   1:  PR[GP1:91,2] = PR[GP1:90,2] + -25.823;
   1:L PR[91] R[100]mm/sec CNT100;
   1:  PR[GP1:91,1] = PR[GP1:90,1] + -0.299;
   1:  PR[GP1:91,2] = PR[GP1:90,2] + -25.163;
   1:L PR[91] R[100]mm/sec CNT100;
   1:  PR[GP1:91,1] = PR[GP1:90,1] + 0.928;
   1:  PR[GP1:91,2] = PR[GP1:90,2] + -24.512;
   1:L PR[91] R[100]mm/sec CNT100;
   1:  PR[GP1:91,1] = PR[GP1:90,1] + 3.642;
   1:  PR[GP1:91,2] = PR[GP1:90,2] + -25.886;
   1:L PR[91] R[100]mm/sec CNT100;
   1:  PR[GP1:91,1] = PR[GP1:90,1] + 4.853;
   1:  PR[GP1:91,2] = PR[GP1:90,2] + -27.292;
   1:L PR[91] R[100]mm/sec CNT100;
   1:  PR[GP1:91,1] = PR[GP1:90,1] + 6.411;
   1:  PR[GP1:91,2] = PR[GP1:90,2] + -28.511;
   1:L PR[91] R[100]mm/sec CNT100;
   1:  PR[GP1:91,1] = PR[GP1:90,1] + 9.247;
   1:  PR[GP1:91,2] = PR[GP1:90,2] + -30.572;
   1:L PR[91] R[100]mm/sec CNT100;
   1:  PR[GP1:91,1] = PR[GP1:90,1] + 13.202;
   1:  PR[GP1:91,2] = PR[GP1:90,2] + -32.635;
   1:L PR[91] R[100]mm/sec CNT100;
   1:  PR[GP1:91,1] = PR[GP1:90,1] + 18.097;
   1:  PR[GP1:91,2] = PR[GP1:90,2] + -34.208;
   1:L PR[91] R[100]mm/sec CNT100;
   1:  PR[GP1:91,1] = PR[GP1:90,1] + 21.818;
   1:  PR[GP1:91,2] = PR[GP1:90,2] + -35.496;
   1:L PR[91] R[100]mm/sec CNT100;
   1:  PR[GP1:91,1] = PR[GP1:90,1] + 27.054;
   1:  PR[GP1:91,2] = PR[GP1:90,2] + -36.185;
   1:L PR[91] R[100]mm/sec CNT100;
   1:  PR[GP1:91,1] = PR[GP1:90,1] + 33.153;
   1:  PR[GP1:91,2] = PR[GP1:90,2] + -35.979;
   1:L PR[91] R[100]mm/sec CNT100;
   1:  PR[GP1:91,1] = PR[GP1:90,1] + 35.421;
   1:  PR[GP1:91,2] = PR[GP1:90,2] + -35.970;
   1:L PR[91] R[100]mm/sec CNT100;
   1:  PR[GP1:91,1] = PR[GP1:90,1] + 41.432;
   1:  PR[GP1:91,2] = PR[GP1:90,2] + -34.676;
   1:L PR[91] R[100]mm/sec CNT100;
   1:  PR[GP1:91,1] = PR[GP1:90,1] + 48.015;
   1:  PR[GP1:91,2] = PR[GP1:90,2] + -32.082;
   1:L PR[91] R[100]mm/sec CNT100;
   1:  PR[GP1:91,1] = PR[GP1:90,1] + 48.422;
   1:  PR[GP1:91,2] = PR[GP1:90,2] + -31.938;
   1:L PR[91] R[100]mm/sec CNT100;
   1:  PR[GP1:91,1] = PR[GP1:90,1] + 54.191;
   1:  PR[GP1:91,2] = PR[GP1:90,2] + -28.371;
   1:L PR[91] R[100]mm/sec CNT100;
   1:  PR[GP1:91,1] = PR[GP1:90,1] + 58.385;
   1:  PR[GP1:91,2] = PR[GP1:90,2] + -24.622;
   1:L PR[91] R[100]mm/sec CNT100;
   1:  PR[GP1:91,1] = PR[GP1:90,1] + 59.664;
   1:  PR[GP1:91,2] = PR[GP1:90,2] + -23.273;
   1:L PR[91] R[100]mm/sec CNT100;
   1:  PR[GP1:91,1] = PR[GP1:90,1] + 62.909;
   1:  PR[GP1:91,2] = PR[GP1:90,2] + -19.073;
   1:L PR[91] R[100]mm/sec CNT100;
   1:  PR[GP1:91,1] = PR[GP1:90,1] + 64.251;
   1:  PR[GP1:91,2] = PR[GP1:90,2] + -16.402;
   1:L PR[91] R[100]mm/sec CNT100;
   1:  PR[GP1:91,1] = PR[GP1:90,1] + 66.515;
   1:  PR[GP1:91,2] = PR[GP1:90,2] + -11.966;
   1:L PR[91] R[100]mm/sec CNT100;
   1:  PR[GP1:91,1] = PR[GP1:90,1] + 67.682;
   1:  PR[GP1:91,2] = PR[GP1:90,2] + -8.056;
   1:L PR[91] R[100]mm/sec CNT100;
   1:  PR[GP1:91,1] = PR[GP1:90,1] + 68.295;
   1:  PR[GP1:91,2] = PR[GP1:90,2] + -4.114;
   1:L PR[91] R[100]mm/sec CNT100;
   1:  PR[GP1:91,1] = PR[GP1:90,1] + 68.664;
   1:  PR[GP1:91,2] = PR[GP1:90,2] + -0.092;
   1:L PR[91] R[100]mm/sec CNT100;
   1:  PR[GP1:91,1] = PR[GP1:90,1] + 68.048;
   1:  PR[GP1:91,2] = PR[GP1:90,2] + 3.822;
   1:L PR[91] R[100]mm/sec CNT100;
   1:  PR[GP1:91,1] = PR[GP1:90,1] + 67.676;
   1:  PR[GP1:91,2] = PR[GP1:90,2] + 7.931;
   1:L PR[91] R[100]mm/sec CNT100;
   1:  PR[GP1:91,1] = PR[GP1:90,1] + 66.514;
   1:  PR[GP1:91,2] = PR[GP1:90,2] + 11.824;
   1:L PR[91] R[100]mm/sec CNT100;
   1:  PR[GP1:91,1] = PR[GP1:90,1] + 65.008;
   1:  PR[GP1:91,2] = PR[GP1:90,2] + 14.824;
   1:L PR[91] R[100]mm/sec CNT100;
   1:  PR[GP1:91,1] = PR[GP1:90,1] + 62.910;
   1:  PR[GP1:91,2] = PR[GP1:90,2] + 18.928;
   1:L PR[91] R[100]mm/sec CNT100;
   1:  PR[GP1:91,1] = PR[GP1:90,1] + 59.664;
   1:  PR[GP1:91,2] = PR[GP1:90,2] + 23.129;
   1:L PR[91] R[100]mm/sec CNT100;
   1:  PR[GP1:91,1] = PR[GP1:90,1] + 58.385;
   1:  PR[GP1:91,2] = PR[GP1:90,2] + 24.478;
   1:L PR[91] R[100]mm/sec CNT100;
   1:  PR[GP1:91,1] = PR[GP1:90,1] + 54.200;
   1:  PR[GP1:91,2] = PR[GP1:90,2] + 28.218;
   1:L PR[91] R[100]mm/sec CNT100;
   1:  PR[GP1:91,1] = PR[GP1:90,1] + 53.739;
   1:  PR[GP1:91,2] = PR[GP1:90,2] + 28.477;
   1:L PR[91] R[100]mm/sec CNT100;
   1:  PR[GP1:91,1] = PR[GP1:90,1] + 51.702;
   1:  PR[GP1:91,2] = PR[GP1:90,2] + 29.761;
   1:L PR[91] R[100]mm/sec CNT100;
   1:  PR[GP1:91,1] = PR[GP1:90,1] + 48.412;
   1:  PR[GP1:91,2] = PR[GP1:90,2] + 31.800;
   1:L PR[91] R[100]mm/sec CNT100;
   1:  PR[GP1:91,1] = PR[GP1:90,1] + 42.606;
   1:  PR[GP1:91,2] = PR[GP1:90,2] + 34.119;
   1:L PR[91] R[100]mm/sec CNT100;
   1:  PR[GP1:91,1] = PR[GP1:90,1] + 41.444;
   1:  PR[GP1:91,2] = PR[GP1:90,2] + 34.529;
   1:L PR[91] R[100]mm/sec CNT100;
   1:  PR[GP1:91,1] = PR[GP1:90,1] + 35.413;
   1:  PR[GP1:91,2] = PR[GP1:90,2] + 35.827;
   1:L PR[91] R[100]mm/sec CNT100;
   1:  PR[GP1:91,1] = PR[GP1:90,1] + 29.973;
   1:  PR[GP1:91,2] = PR[GP1:90,2] + 36.032;
   1:L PR[91] R[100]mm/sec CNT100;
   1:  PR[GP1:91,1] = PR[GP1:90,1] + 27.067;
   1:  PR[GP1:91,2] = PR[GP1:90,2] + 36.043;
   1:L PR[91] R[100]mm/sec CNT100;
   1:  PR[GP1:91,1] = PR[GP1:90,1] + 21.816;
   1:  PR[GP1:91,2] = PR[GP1:90,2] + 35.352;
   1:L PR[91] R[100]mm/sec CNT100;
   1:  PR[GP1:91,1] = PR[GP1:90,1] + 17.313;
   1:  PR[GP1:91,2] = PR[GP1:90,2] + 33.919;
   1:L PR[91] R[100]mm/sec CNT100;
   1:  PR[GP1:91,1] = PR[GP1:90,1] + 13.215;
   1:  PR[GP1:91,2] = PR[GP1:90,2] + 32.499;
   1:L PR[91] R[100]mm/sec CNT100;
   1:  PR[GP1:91,1] = PR[GP1:90,1] + 9.248;
   1:  PR[GP1:91,2] = PR[GP1:90,2] + 30.428;
   1:L PR[91] R[100]mm/sec CNT100;
   1:  PR[GP1:91,1] = PR[GP1:90,1] + 7.195;
   1:  PR[GP1:91,2] = PR[GP1:90,2] + 28.978;
   1:L PR[91] R[100]mm/sec CNT100;
   1:  PR[GP1:91,1] = PR[GP1:90,1] + 5.201;
   1:  PR[GP1:91,2] = PR[GP1:90,2] + 27.418;
   1:L PR[91] R[100]mm/sec CNT100;
   1:  PR[GP1:91,1] = PR[GP1:90,1] + 3.626;
   1:  PR[GP1:91,2] = PR[GP1:90,2] + 25.585;
   1:L PR[91] R[100]mm/sec CNT100;
   1:  PR[GP1:91,1] = PR[GP1:90,1] + 2.246;
   1:  PR[GP1:91,2] = PR[GP1:90,2] + 25.040;
   1:L PR[91] R[100]mm/sec CNT100;
   1:  PR[GP1:91,1] = PR[GP1:90,1] + 1.042;
   1:  PR[GP1:91,2] = PR[GP1:90,2] + 24.425;
   1:L PR[91] R[100]mm/sec CNT100;
   1:  ! -- Layer/Ebene 83 -- !;
   1:  PR[91] = PR[90];
   1:  PR[GP1:91,1] = PR[GP1:90,1] + -1.921;
   1:  PR[GP1:91,2] = PR[GP1:90,2] + 25.141;
   1:  PR[GP1:91,3] = PR[GP1:90,3] + 50.935;
   1:L PR[91] R[100]mm/sec CNT100;
   1:  PR[GP1:91,1] = PR[GP1:90,1] + -3.401;
   1:  PR[GP1:91,2] = PR[GP1:90,2] + 25.893;
   1:L PR[91] R[100]mm/sec CNT100;
   1:  PR[GP1:91,1] = PR[GP1:90,1] + -4.816;
   1:  PR[GP1:91,2] = PR[GP1:90,2] + 27.539;
   1:L PR[91] R[100]mm/sec CNT100;
   1:  PR[GP1:91,1] = PR[GP1:90,1] + -6.646;
   1:  PR[GP1:91,2] = PR[GP1:90,2] + 28.972;
   1:L PR[91] R[100]mm/sec CNT100;
   1:  PR[GP1:91,1] = PR[GP1:90,1] + -8.813;
   1:  PR[GP1:91,2] = PR[GP1:90,2] + 30.503;
   1:L PR[91] R[100]mm/sec CNT100;
   1:  PR[GP1:91,1] = PR[GP1:90,1] + -12.667;
   1:  PR[GP1:91,2] = PR[GP1:90,2] + 32.519;
   1:L PR[91] R[100]mm/sec CNT100;
   1:  PR[GP1:91,1] = PR[GP1:90,1] + -17.399;
   1:  PR[GP1:91,2] = PR[GP1:90,2] + 34.040;
   1:L PR[91] R[100]mm/sec CNT100;
   1:  PR[GP1:91,1] = PR[GP1:90,1] + -21.417;
   1:  PR[GP1:91,2] = PR[GP1:90,2] + 35.429;
   1:L PR[91] R[100]mm/sec CNT100;
   1:  PR[GP1:91,1] = PR[GP1:90,1] + -26.506;
   1:  PR[GP1:91,2] = PR[GP1:90,2] + 36.094;
   1:L PR[91] R[100]mm/sec CNT100;
   1:  PR[GP1:91,1] = PR[GP1:90,1] + -32.458;
   1:  PR[GP1:91,2] = PR[GP1:90,2] + 35.889;
   1:L PR[91] R[100]mm/sec CNT100;
   1:  PR[GP1:91,1] = PR[GP1:90,1] + -35.059;
   1:  PR[GP1:91,2] = PR[GP1:90,2] + 35.876;
   1:L PR[91] R[100]mm/sec CNT100;
   1:  PR[GP1:91,1] = PR[GP1:90,1] + -40.921;
   1:  PR[GP1:91,2] = PR[GP1:90,2] + 34.612;
   1:L PR[91] R[100]mm/sec CNT100;
   1:  PR[GP1:91,1] = PR[GP1:90,1] + -47.325;
   1:  PR[GP1:91,2] = PR[GP1:90,2] + 32.076;
   1:L PR[91] R[100]mm/sec CNT100;
   1:  PR[GP1:91,1] = PR[GP1:90,1] + -48.060;
   1:  PR[GP1:91,2] = PR[GP1:90,2] + 31.815;
   1:L PR[91] R[100]mm/sec CNT100;
   1:  PR[GP1:91,1] = PR[GP1:90,1] + -53.826;
   1:  PR[GP1:91,2] = PR[GP1:90,2] + 28.224;
   1:L PR[91] R[100]mm/sec CNT100;
   1:  PR[GP1:91,1] = PR[GP1:90,1] + -58.292;
   1:  PR[GP1:91,2] = PR[GP1:90,2] + 24.219;
   1:L PR[91] R[100]mm/sec CNT100;
   1:  PR[GP1:91,1] = PR[GP1:90,1] + -59.159;
   1:  PR[GP1:91,2] = PR[GP1:90,2] + 23.308;
   1:L PR[91] R[100]mm/sec CNT100;
   1:  PR[GP1:91,1] = PR[GP1:90,1] + -62.600;
   1:  PR[GP1:91,2] = PR[GP1:90,2] + 18.843;
   1:L PR[91] R[100]mm/sec CNT100;
   1:  PR[GP1:91,1] = PR[GP1:90,1] + -66.103;
   1:  PR[GP1:91,2] = PR[GP1:90,2] + 11.880;
   1:L PR[91] R[100]mm/sec CNT100;
   1:  PR[GP1:91,1] = PR[GP1:90,1] + -67.370;
   1:  PR[GP1:91,2] = PR[GP1:90,2] + 7.576;
   1:L PR[91] R[100]mm/sec CNT100;
   1:  PR[GP1:91,1] = PR[GP1:90,1] + -67.893;
   1:  PR[GP1:91,2] = PR[GP1:90,2] + 4.221;
   1:L PR[91] R[100]mm/sec CNT100;
   1:  PR[GP1:91,1] = PR[GP1:90,1] + -68.277;
   1:  PR[GP1:91,2] = PR[GP1:90,2] + -0.052;
   1:L PR[91] R[100]mm/sec CNT100;
   1:  PR[GP1:91,1] = PR[GP1:90,1] + -67.748;
   1:  PR[GP1:91,2] = PR[GP1:90,2] + -3.402;
   1:L PR[91] R[100]mm/sec CNT100;
   1:  PR[GP1:91,1] = PR[GP1:90,1] + -67.364;
   1:  PR[GP1:91,2] = PR[GP1:90,2] + -7.739;
   1:L PR[91] R[100]mm/sec CNT100;
   1:  PR[GP1:91,1] = PR[GP1:90,1] + -66.103;
   1:  PR[GP1:91,2] = PR[GP1:90,2] + -12.024;
   1:L PR[91] R[100]mm/sec CNT100;
   1:  PR[GP1:91,1] = PR[GP1:90,1] + -62.600;
   1:  PR[GP1:91,2] = PR[GP1:90,2] + -18.987;
   1:L PR[91] R[100]mm/sec CNT100;
   1:  PR[GP1:91,1] = PR[GP1:90,1] + -59.159;
   1:  PR[GP1:91,2] = PR[GP1:90,2] + -23.452;
   1:L PR[91] R[100]mm/sec CNT100;
   1:  PR[GP1:91,1] = PR[GP1:90,1] + -58.292;
   1:  PR[GP1:91,2] = PR[GP1:90,2] + -24.363;
   1:L PR[91] R[100]mm/sec CNT100;
   1:  PR[GP1:91,1] = PR[GP1:90,1] + -53.826;
   1:  PR[GP1:91,2] = PR[GP1:90,2] + -28.368;
   1:L PR[91] R[100]mm/sec CNT100;
   1:  PR[GP1:91,1] = PR[GP1:90,1] + -48.048;
   1:  PR[GP1:91,2] = PR[GP1:90,2] + -31.966;
   1:L PR[91] R[100]mm/sec CNT100;
   1:  PR[GP1:91,1] = PR[GP1:90,1] + -42.387;
   1:  PR[GP1:91,2] = PR[GP1:90,2] + -34.239;
   1:L PR[91] R[100]mm/sec CNT100;
   1:  PR[GP1:91,1] = PR[GP1:90,1] + -40.930;
   1:  PR[GP1:91,2] = PR[GP1:90,2] + -34.754;
   1:L PR[91] R[100]mm/sec CNT100;
   1:  PR[GP1:91,1] = PR[GP1:90,1] + -35.047;
   1:  PR[GP1:91,2] = PR[GP1:90,2] + -36.023;
   1:L PR[91] R[100]mm/sec CNT100;
   1:  PR[GP1:91,1] = PR[GP1:90,1] + -29.722;
   1:  PR[GP1:91,2] = PR[GP1:90,2] + -36.228;
   1:L PR[91] R[100]mm/sec CNT100;
   1:  PR[GP1:91,1] = PR[GP1:90,1] + -26.510;
   1:  PR[GP1:91,2] = PR[GP1:90,2] + -36.238;
   1:L PR[91] R[100]mm/sec CNT100;
   1:  PR[GP1:91,1] = PR[GP1:90,1] + -21.403;
   1:  PR[GP1:91,2] = PR[GP1:90,2] + -35.571;
   1:L PR[91] R[100]mm/sec CNT100;
   1:  PR[GP1:91,1] = PR[GP1:90,1] + -17.035;
   1:  PR[GP1:91,2] = PR[GP1:90,2] + -34.181;
   1:L PR[91] R[100]mm/sec CNT100;
   1:  PR[GP1:91,1] = PR[GP1:90,1] + -12.666;
   1:  PR[GP1:91,2] = PR[GP1:90,2] + -32.663;
   1:L PR[91] R[100]mm/sec CNT100;
   1:  PR[GP1:91,1] = PR[GP1:90,1] + -8.812;
   1:  PR[GP1:91,2] = PR[GP1:90,2] + -30.646;
   1:L PR[91] R[100]mm/sec CNT100;
   1:  PR[GP1:91,1] = PR[GP1:90,1] + -5.818;
   1:  PR[GP1:91,2] = PR[GP1:90,2] + -28.471;
   1:L PR[91] R[100]mm/sec CNT100;
   1:  PR[GP1:91,1] = PR[GP1:90,1] + -4.454;
   1:  PR[GP1:91,2] = PR[GP1:90,2] + -27.403;
   1:L PR[91] R[100]mm/sec CNT100;
   1:  PR[GP1:91,1] = PR[GP1:90,1] + -3.344;
   1:  PR[GP1:91,2] = PR[GP1:90,2] + -26.115;
   1:L PR[91] R[100]mm/sec CNT100;
   1:  PR[GP1:91,1] = PR[GP1:90,1] + -0.132;
   1:  PR[GP1:91,2] = PR[GP1:90,2] + -25.426;
   1:L PR[91] R[100]mm/sec CNT100;
   1:  PR[GP1:91,1] = PR[GP1:90,1] + 0.970;
   1:  PR[GP1:91,2] = PR[GP1:90,2] + -24.842;
   1:L PR[91] R[100]mm/sec CNT100;
   1:  PR[GP1:91,1] = PR[GP1:90,1] + 3.612;
   1:  PR[GP1:91,2] = PR[GP1:90,2] + -26.179;
   1:L PR[91] R[100]mm/sec CNT100;
   1:  PR[GP1:91,1] = PR[GP1:90,1] + 4.677;
   1:  PR[GP1:91,2] = PR[GP1:90,2] + -27.416;
   1:L PR[91] R[100]mm/sec CNT100;
   1:  PR[GP1:91,1] = PR[GP1:90,1] + 6.035;
   1:  PR[GP1:91,2] = PR[GP1:90,2] + -28.479;
   1:L PR[91] R[100]mm/sec CNT100;
   1:  PR[GP1:91,1] = PR[GP1:90,1] + 9.035;
   1:  PR[GP1:91,2] = PR[GP1:90,2] + -30.658;
   1:L PR[91] R[100]mm/sec CNT100;
   1:  PR[GP1:91,1] = PR[GP1:90,1] + 12.860;
   1:  PR[GP1:91,2] = PR[GP1:90,2] + -32.654;
   1:L PR[91] R[100]mm/sec CNT100;
   1:  PR[GP1:91,1] = PR[GP1:90,1] + 17.596;
   1:  PR[GP1:91,2] = PR[GP1:90,2] + -34.176;
   1:L PR[91] R[100]mm/sec CNT100;
   1:  PR[GP1:91,1] = PR[GP1:90,1] + 21.619;
   1:  PR[GP1:91,2] = PR[GP1:90,2] + -35.568;
   1:L PR[91] R[100]mm/sec CNT100;
   1:  PR[GP1:91,1] = PR[GP1:90,1] + 26.702;
   1:  PR[GP1:91,2] = PR[GP1:90,2] + -36.237;
   1:L PR[91] R[100]mm/sec CNT100;
   1:  PR[GP1:91,1] = PR[GP1:90,1] + 32.625;
   1:  PR[GP1:91,2] = PR[GP1:90,2] + -36.038;
   1:L PR[91] R[100]mm/sec CNT100;
   1:  PR[GP1:91,1] = PR[GP1:90,1] + 35.233;
   1:  PR[GP1:91,2] = PR[GP1:90,2] + -36.026;
   1:L PR[91] R[100]mm/sec CNT100;
   1:  PR[GP1:91,1] = PR[GP1:90,1] + 41.087;
   1:  PR[GP1:91,2] = PR[GP1:90,2] + -34.766;
   1:L PR[91] R[100]mm/sec CNT100;
   1:  PR[GP1:91,1] = PR[GP1:90,1] + 47.499;
   1:  PR[GP1:91,2] = PR[GP1:90,2] + -32.240;
   1:L PR[91] R[100]mm/sec CNT100;
   1:  PR[GP1:91,1] = PR[GP1:90,1] + 48.239;
   1:  PR[GP1:91,2] = PR[GP1:90,2] + -31.978;
   1:L PR[91] R[100]mm/sec CNT100;
   1:  PR[GP1:91,1] = PR[GP1:90,1] + 53.973;
   1:  PR[GP1:91,2] = PR[GP1:90,2] + -28.424;
   1:L PR[91] R[100]mm/sec CNT100;
   1:  PR[GP1:91,1] = PR[GP1:90,1] + 58.437;
   1:  PR[GP1:91,2] = PR[GP1:90,2] + -24.434;
   1:L PR[91] R[100]mm/sec CNT100;
   1:  PR[GP1:91,1] = PR[GP1:90,1] + 59.292;
   1:  PR[GP1:91,2] = PR[GP1:90,2] + -23.533;
   1:L PR[91] R[100]mm/sec CNT100;
   1:  PR[GP1:91,1] = PR[GP1:90,1] + 62.782;
   1:  PR[GP1:91,2] = PR[GP1:90,2] + -19.015;
   1:L PR[91] R[100]mm/sec CNT100;
   1:  PR[GP1:91,1] = PR[GP1:90,1] + 63.841;
   1:  PR[GP1:91,2] = PR[GP1:90,2] + -16.908;
   1:L PR[91] R[100]mm/sec CNT100;
   1:  PR[GP1:91,1] = PR[GP1:90,1] + 66.297;
   1:  PR[GP1:91,2] = PR[GP1:90,2] + -12.096;
   1:L PR[91] R[100]mm/sec CNT100;
   1:  PR[GP1:91,1] = PR[GP1:90,1] + 67.564;
   1:  PR[GP1:91,2] = PR[GP1:90,2] + -7.850;
   1:L PR[91] R[100]mm/sec CNT100;
   1:  PR[GP1:91,1] = PR[GP1:90,1] + 68.087;
   1:  PR[GP1:91,2] = PR[GP1:90,2] + -4.488;
   1:L PR[91] R[100]mm/sec CNT100;
   1:  PR[GP1:91,1] = PR[GP1:90,1] + 68.490;
   1:  PR[GP1:91,2] = PR[GP1:90,2] + -0.092;
   1:L PR[91] R[100]mm/sec CNT100;
   1:  PR[GP1:91,1] = PR[GP1:90,1] + 67.961;
   1:  PR[GP1:91,2] = PR[GP1:90,2] + 3.267;
   1:L PR[91] R[100]mm/sec CNT100;
   1:  PR[GP1:91,1] = PR[GP1:90,1] + 67.558;
   1:  PR[GP1:91,2] = PR[GP1:90,2] + 7.724;
   1:L PR[91] R[100]mm/sec CNT100;
   1:  PR[GP1:91,1] = PR[GP1:90,1] + 66.296;
   1:  PR[GP1:91,2] = PR[GP1:90,2] + 11.954;
   1:L PR[91] R[100]mm/sec CNT100;
   1:  PR[GP1:91,1] = PR[GP1:90,1] + 65.040;
   1:  PR[GP1:91,2] = PR[GP1:90,2] + 14.456;
   1:L PR[91] R[100]mm/sec CNT100;
   1:  PR[GP1:91,1] = PR[GP1:90,1] + 62.784;
   1:  PR[GP1:91,2] = PR[GP1:90,2] + 18.870;
   1:L PR[91] R[100]mm/sec CNT100;
   1:  PR[GP1:91,1] = PR[GP1:90,1] + 59.292;
   1:  PR[GP1:91,2] = PR[GP1:90,2] + 23.389;
   1:L PR[91] R[100]mm/sec CNT100;
   1:  PR[GP1:91,1] = PR[GP1:90,1] + 58.437;
   1:  PR[GP1:91,2] = PR[GP1:90,2] + 24.290;
   1:L PR[91] R[100]mm/sec CNT100;
   1:  PR[GP1:91,1] = PR[GP1:90,1] + 53.973;
   1:  PR[GP1:91,2] = PR[GP1:90,2] + 28.280;
   1:L PR[91] R[100]mm/sec CNT100;
   1:  PR[GP1:91,1] = PR[GP1:90,1] + 48.230;
   1:  PR[GP1:91,2] = PR[GP1:90,2] + 31.840;
   1:L PR[91] R[100]mm/sec CNT100;
   1:  PR[GP1:91,1] = PR[GP1:90,1] + 42.561;
   1:  PR[GP1:91,2] = PR[GP1:90,2] + 34.104;
   1:L PR[91] R[100]mm/sec CNT100;
   1:  PR[GP1:91,1] = PR[GP1:90,1] + 41.099;
   1:  PR[GP1:91,2] = PR[GP1:90,2] + 34.620;
   1:L PR[91] R[100]mm/sec CNT100;
   1:  PR[GP1:91,1] = PR[GP1:90,1] + 35.226;
   1:  PR[GP1:91,2] = PR[GP1:90,2] + 35.884;
   1:L PR[91] R[100]mm/sec CNT100;
   1:  PR[GP1:91,1] = PR[GP1:90,1] + 29.928;
   1:  PR[GP1:91,2] = PR[GP1:90,2] + 36.084;
   1:L PR[91] R[100]mm/sec CNT100;
   1:  PR[GP1:91,1] = PR[GP1:90,1] + 26.716;
   1:  PR[GP1:91,2] = PR[GP1:90,2] + 36.095;
   1:L PR[91] R[100]mm/sec CNT100;
   1:  PR[GP1:91,1] = PR[GP1:90,1] + 21.618;
   1:  PR[GP1:91,2] = PR[GP1:90,2] + 35.425;
   1:L PR[91] R[100]mm/sec CNT100;
   1:  PR[GP1:91,1] = PR[GP1:90,1] + 17.245;
   1:  PR[GP1:91,2] = PR[GP1:90,2] + 34.033;
   1:L PR[91] R[100]mm/sec CNT100;
   1:  PR[GP1:91,1] = PR[GP1:90,1] + 12.873;
   1:  PR[GP1:91,2] = PR[GP1:90,2] + 32.517;
   1:L PR[91] R[100]mm/sec CNT100;
   1:  PR[GP1:91,1] = PR[GP1:90,1] + 9.036;
   1:  PR[GP1:91,2] = PR[GP1:90,2] + 30.515;
   1:L PR[91] R[100]mm/sec CNT100;
   1:  PR[GP1:91,1] = PR[GP1:90,1] + 6.864;
   1:  PR[GP1:91,2] = PR[GP1:90,2] + 28.981;
   1:L PR[91] R[100]mm/sec CNT100;
   1:  PR[GP1:91,1] = PR[GP1:90,1] + 5.043;
   1:  PR[GP1:91,2] = PR[GP1:90,2] + 27.556;
   1:L PR[91] R[100]mm/sec CNT100;
   1:  PR[GP1:91,1] = PR[GP1:90,1] + 3.596;
   1:  PR[GP1:91,2] = PR[GP1:90,2] + 25.871;
   1:L PR[91] R[100]mm/sec CNT100;
   1:  PR[GP1:91,1] = PR[GP1:90,1] + 2.158;
   1:  PR[GP1:91,2] = PR[GP1:90,2] + 25.303;
   1:L PR[91] R[100]mm/sec CNT100;
   1:  PR[GP1:91,1] = PR[GP1:90,1] + 1.084;
   1:  PR[GP1:91,2] = PR[GP1:90,2] + 24.754;
   1:L PR[91] R[100]mm/sec CNT100;
   1:  ! -- Layer/Ebene 84 -- !;
   1:  PR[91] = PR[90];
   1:  PR[GP1:91,1] = PR[GP1:90,1] + -2.010;
   1:  PR[GP1:91,2] = PR[GP1:90,2] + 25.487;
   1:  PR[GP1:91,3] = PR[GP1:90,3] + 51.545;
   1:L PR[91] R[100]mm/sec CNT100;
   1:  PR[GP1:91,1] = PR[GP1:90,1] + -3.372;
   1:  PR[GP1:91,2] = PR[GP1:90,2] + 26.180;
   1:L PR[91] R[100]mm/sec CNT100;
   1:  PR[GP1:91,1] = PR[GP1:90,1] + -4.660;
   1:  PR[GP1:91,2] = PR[GP1:90,2] + 27.678;
   1:L PR[91] R[100]mm/sec CNT100;
   1:  PR[GP1:91,1] = PR[GP1:90,1] + -6.317;
   1:  PR[GP1:91,2] = PR[GP1:90,2] + 28.975;
   1:L PR[91] R[100]mm/sec CNT100;
   1:  PR[GP1:91,1] = PR[GP1:90,1] + -8.602;
   1:  PR[GP1:91,2] = PR[GP1:90,2] + 30.590;
   1:L PR[91] R[100]mm/sec CNT100;
   1:  PR[GP1:91,1] = PR[GP1:90,1] + -12.325;
   1:  PR[GP1:91,2] = PR[GP1:90,2] + 32.538;
   1:L PR[91] R[100]mm/sec CNT100;
   1:  PR[GP1:91,1] = PR[GP1:90,1] + -16.898;
   1:  PR[GP1:91,2] = PR[GP1:90,2] + 34.007;
   1:L PR[91] R[100]mm/sec CNT100;
   1:  PR[GP1:91,1] = PR[GP1:90,1] + -21.218;
   1:  PR[GP1:91,2] = PR[GP1:90,2] + 35.501;
   1:L PR[91] R[100]mm/sec CNT100;
   1:  PR[GP1:91,1] = PR[GP1:90,1] + -26.155;
   1:  PR[GP1:91,2] = PR[GP1:90,2] + 36.146;
   1:L PR[91] R[100]mm/sec CNT100;
   1:  PR[GP1:91,1] = PR[GP1:90,1] + -31.929;
   1:  PR[GP1:91,2] = PR[GP1:90,2] + 35.947;
   1:L PR[91] R[100]mm/sec CNT100;
   1:  PR[GP1:91,1] = PR[GP1:90,1] + -34.872;
   1:  PR[GP1:91,2] = PR[GP1:90,2] + 35.933;
   1:L PR[91] R[100]mm/sec CNT100;
   1:  PR[GP1:91,1] = PR[GP1:90,1] + -40.575;
   1:  PR[GP1:91,2] = PR[GP1:90,2] + 34.702;
   1:L PR[91] R[100]mm/sec CNT100;
   1:  PR[GP1:91,1] = PR[GP1:90,1] + -46.809;
   1:  PR[GP1:91,2] = PR[GP1:90,2] + 32.234;
   1:L PR[91] R[100]mm/sec CNT100;
   1:  PR[GP1:91,1] = PR[GP1:90,1] + -47.876;
   1:  PR[GP1:91,2] = PR[GP1:90,2] + 31.855;
   1:L PR[91] R[100]mm/sec CNT100;
   1:  PR[GP1:91,1] = PR[GP1:90,1] + -53.508;
   1:  PR[GP1:91,2] = PR[GP1:90,2] + 28.347;
   1:L PR[91] R[100]mm/sec CNT100;
   1:  PR[GP1:91,1] = PR[GP1:90,1] + -55.883;
   1:  PR[GP1:91,2] = PR[GP1:90,2] + 26.238;
   1:L PR[91] R[100]mm/sec CNT100;
   1:  PR[GP1:91,1] = PR[GP1:90,1] + -58.348;
   1:  PR[GP1:91,2] = PR[GP1:90,2] + 24.028;
   1:L PR[91] R[100]mm/sec CNT100;
   1:  PR[GP1:91,1] = PR[GP1:90,1] + -58.792;
   1:  PR[GP1:91,2] = PR[GP1:90,2] + 23.562;
   1:L PR[91] R[100]mm/sec CNT100;
   1:  PR[GP1:91,1] = PR[GP1:90,1] + -62.475;
   1:  PR[GP1:91,2] = PR[GP1:90,2] + 18.782;
   1:L PR[91] R[100]mm/sec CNT100;
   1:  PR[GP1:91,1] = PR[GP1:90,1] + -65.886;
   1:  PR[GP1:91,2] = PR[GP1:90,2] + 12.006;
   1:L PR[91] R[100]mm/sec CNT100;
   1:  PR[GP1:91,1] = PR[GP1:90,1] + -67.253;
   1:  PR[GP1:91,2] = PR[GP1:90,2] + 7.362;
   1:L PR[91] R[100]mm/sec CNT100;
   1:  PR[GP1:91,1] = PR[GP1:90,1] + -67.686;
   1:  PR[GP1:91,2] = PR[GP1:90,2] + 4.584;
   1:L PR[91] R[100]mm/sec CNT100;
   1:  PR[GP1:91,1] = PR[GP1:90,1] + -68.103;
   1:  PR[GP1:91,2] = PR[GP1:90,2] + -0.052;
   1:L PR[91] R[100]mm/sec CNT100;
   1:  PR[GP1:91,1] = PR[GP1:90,1] + -67.661;
   1:  PR[GP1:91,2] = PR[GP1:90,2] + -2.849;
   1:L PR[91] R[100]mm/sec CNT100;
   1:  PR[GP1:91,1] = PR[GP1:90,1] + -67.248;
   1:  PR[GP1:91,2] = PR[GP1:90,2] + -7.525;
   1:L PR[91] R[100]mm/sec CNT100;
   1:  PR[GP1:91,1] = PR[GP1:90,1] + -65.886;
   1:  PR[GP1:91,2] = PR[GP1:90,2] + -12.150;
   1:L PR[91] R[100]mm/sec CNT100;
   1:  PR[GP1:91,1] = PR[GP1:90,1] + -62.475;
   1:  PR[GP1:91,2] = PR[GP1:90,2] + -18.926;
   1:L PR[91] R[100]mm/sec CNT100;
   1:  PR[GP1:91,1] = PR[GP1:90,1] + -58.792;
   1:  PR[GP1:91,2] = PR[GP1:90,2] + -23.706;
   1:L PR[91] R[100]mm/sec CNT100;
   1:  PR[GP1:91,1] = PR[GP1:90,1] + -58.348;
   1:  PR[GP1:91,2] = PR[GP1:90,2] + -24.172;
   1:L PR[91] R[100]mm/sec CNT100;
   1:  PR[GP1:91,1] = PR[GP1:90,1] + -53.720;
   1:  PR[GP1:91,2] = PR[GP1:90,2] + -28.322;
   1:L PR[91] R[100]mm/sec CNT100;
   1:  PR[GP1:91,1] = PR[GP1:90,1] + -53.520;
   1:  PR[GP1:91,2] = PR[GP1:90,2] + -28.483;
   1:L PR[91] R[100]mm/sec CNT100;
   1:  PR[GP1:91,1] = PR[GP1:90,1] + -47.865;
   1:  PR[GP1:91,2] = PR[GP1:90,2] + -32.006;
   1:L PR[91] R[100]mm/sec CNT100;
   1:  PR[GP1:91,1] = PR[GP1:90,1] + -42.341;
   1:  PR[GP1:91,2] = PR[GP1:90,2] + -34.224;
   1:L PR[91] R[100]mm/sec CNT100;
   1:  PR[GP1:91,1] = PR[GP1:90,1] + -40.584;
   1:  PR[GP1:91,2] = PR[GP1:90,2] + -34.844;
   1:L PR[91] R[100]mm/sec CNT100;
   1:  PR[GP1:91,1] = PR[GP1:90,1] + -34.858;
   1:  PR[GP1:91,2] = PR[GP1:90,2] + -36.079;
   1:L PR[91] R[100]mm/sec CNT100;
   1:  PR[GP1:91,1] = PR[GP1:90,1] + -29.676;
   1:  PR[GP1:91,2] = PR[GP1:90,2] + -36.279;
   1:L PR[91] R[100]mm/sec CNT100;
   1:  PR[GP1:91,1] = PR[GP1:90,1] + -26.158;
   1:  PR[GP1:91,2] = PR[GP1:90,2] + -36.290;
   1:L PR[91] R[100]mm/sec CNT100;
   1:  PR[GP1:91,1] = PR[GP1:90,1] + -21.204;
   1:  PR[GP1:91,2] = PR[GP1:90,2] + -35.643;
   1:L PR[91] R[100]mm/sec CNT100;
   1:  PR[GP1:91,1] = PR[GP1:90,1] + -16.967;
   1:  PR[GP1:91,2] = PR[GP1:90,2] + -34.294;
   1:L PR[91] R[100]mm/sec CNT100;
   1:  PR[GP1:91,1] = PR[GP1:90,1] + -12.324;
   1:  PR[GP1:91,2] = PR[GP1:90,2] + -32.681;
   1:L PR[91] R[100]mm/sec CNT100;
   1:  PR[GP1:91,1] = PR[GP1:90,1] + -8.601;
   1:  PR[GP1:91,2] = PR[GP1:90,2] + -30.733;
   1:L PR[91] R[100]mm/sec CNT100;
   1:  PR[GP1:91,1] = PR[GP1:90,1] + -5.444;
   1:  PR[GP1:91,2] = PR[GP1:90,2] + -28.440;
   1:L PR[91] R[100]mm/sec CNT100;
   1:  PR[GP1:91,1] = PR[GP1:90,1] + -4.281;
   1:  PR[GP1:91,2] = PR[GP1:90,2] + -27.529;
   1:L PR[91] R[100]mm/sec CNT100;
   1:  PR[GP1:91,1] = PR[GP1:90,1] + -3.315;
   1:  PR[GP1:91,2] = PR[GP1:90,2] + -26.408;
   1:L PR[91] R[100]mm/sec CNT100;
   1:  PR[GP1:91,1] = PR[GP1:90,1] + 0.035;
   1:  PR[GP1:91,2] = PR[GP1:90,2] + -25.689;
   1:L PR[91] R[100]mm/sec CNT100;
   1:  PR[GP1:91,1] = PR[GP1:90,1] + 1.011;
   1:  PR[GP1:91,2] = PR[GP1:90,2] + -25.172;
   1:L PR[91] R[100]mm/sec CNT100;
   1:  PR[GP1:91,1] = PR[GP1:90,1] + 3.582;
   1:  PR[GP1:91,2] = PR[GP1:90,2] + -26.472;
   1:L PR[91] R[100]mm/sec CNT100;
   1:  PR[GP1:91,1] = PR[GP1:90,1] + 4.502;
   1:  PR[GP1:91,2] = PR[GP1:90,2] + -27.541;
   1:L PR[91] R[100]mm/sec CNT100;
   1:  PR[GP1:91,1] = PR[GP1:90,1] + 5.660;
   1:  PR[GP1:91,2] = PR[GP1:90,2] + -28.447;
   1:L PR[91] R[100]mm/sec CNT100;
   1:  PR[GP1:91,1] = PR[GP1:90,1] + 8.824;
   1:  PR[GP1:91,2] = PR[GP1:90,2] + -30.745;
   1:L PR[91] R[100]mm/sec CNT100;
   1:  PR[GP1:91,1] = PR[GP1:90,1] + 12.517;
   1:  PR[GP1:91,2] = PR[GP1:90,2] + -32.673;
   1:L PR[91] R[100]mm/sec CNT100;
   1:  PR[GP1:91,1] = PR[GP1:90,1] + 17.094;
   1:  PR[GP1:91,2] = PR[GP1:90,2] + -34.143;
   1:L PR[91] R[100]mm/sec CNT100;
   1:  PR[GP1:91,1] = PR[GP1:90,1] + 21.420;
   1:  PR[GP1:91,2] = PR[GP1:90,2] + -35.641;
   1:L PR[91] R[100]mm/sec CNT100;
   1:  PR[GP1:91,1] = PR[GP1:90,1] + 26.350;
   1:  PR[GP1:91,2] = PR[GP1:90,2] + -36.289;
   1:L PR[91] R[100]mm/sec CNT100;
   1:  PR[GP1:91,1] = PR[GP1:90,1] + 32.098;
   1:  PR[GP1:91,2] = PR[GP1:90,2] + -36.096;
   1:L PR[91] R[100]mm/sec CNT100;
   1:  PR[GP1:91,1] = PR[GP1:90,1] + 35.046;
   1:  PR[GP1:91,2] = PR[GP1:90,2] + -36.083;
   1:L PR[91] R[100]mm/sec CNT100;
   1:  PR[GP1:91,1] = PR[GP1:90,1] + 40.742;
   1:  PR[GP1:91,2] = PR[GP1:90,2] + -34.857;
   1:L PR[91] R[100]mm/sec CNT100;
   1:  PR[GP1:91,1] = PR[GP1:90,1] + 46.984;
   1:  PR[GP1:91,2] = PR[GP1:90,2] + -32.397;
   1:L PR[91] R[100]mm/sec CNT100;
   1:  PR[GP1:91,1] = PR[GP1:90,1] + 48.056;
   1:  PR[GP1:91,2] = PR[GP1:90,2] + -32.017;
   1:L PR[91] R[100]mm/sec CNT100;
   1:  PR[GP1:91,1] = PR[GP1:90,1] + 53.654;
   1:  PR[GP1:91,2] = PR[GP1:90,2] + -28.548;
   1:L PR[91] R[100]mm/sec CNT100;
   1:  PR[GP1:91,1] = PR[GP1:90,1] + 58.489;
   1:  PR[GP1:91,2] = PR[GP1:90,2] + -24.246;
   1:L PR[91] R[100]mm/sec CNT100;
   1:  PR[GP1:91,1] = PR[GP1:90,1] + 58.919;
   1:  PR[GP1:91,2] = PR[GP1:90,2] + -23.793;
   1:L PR[91] R[100]mm/sec CNT100;
   1:  PR[GP1:91,1] = PR[GP1:90,1] + 62.656;
   1:  PR[GP1:91,2] = PR[GP1:90,2] + -18.956;
   1:L PR[91] R[100]mm/sec CNT100;
   1:  PR[GP1:91,1] = PR[GP1:90,1] + 66.078;
   1:  PR[GP1:91,2] = PR[GP1:90,2] + -12.226;
   1:L PR[91] R[100]mm/sec CNT100;
   1:  PR[GP1:91,1] = PR[GP1:90,1] + 67.446;
   1:  PR[GP1:91,2] = PR[GP1:90,2] + -7.644;
   1:L PR[91] R[100]mm/sec CNT100;
   1:  PR[GP1:91,1] = PR[GP1:90,1] + 67.878;
   1:  PR[GP1:91,2] = PR[GP1:90,2] + -4.861;
   1:L PR[91] R[100]mm/sec CNT100;
   1:  PR[GP1:91,1] = PR[GP1:90,1] + 68.316;
   1:  PR[GP1:91,2] = PR[GP1:90,2] + -0.092;
   1:L PR[91] R[100]mm/sec CNT100;
   1:  PR[GP1:91,1] = PR[GP1:90,1] + 67.875;
   1:  PR[GP1:91,2] = PR[GP1:90,2] + 2.713;
   1:L PR[91] R[100]mm/sec CNT100;
   1:  PR[GP1:91,1] = PR[GP1:90,1] + 67.440;
   1:  PR[GP1:91,2] = PR[GP1:90,2] + 7.518;
   1:L PR[91] R[100]mm/sec CNT100;
   1:  PR[GP1:91,1] = PR[GP1:90,1] + 66.078;
   1:  PR[GP1:91,2] = PR[GP1:90,2] + 12.084;
   1:L PR[91] R[100]mm/sec CNT100;
   1:  PR[GP1:91,1] = PR[GP1:90,1] + 65.071;
   1:  PR[GP1:91,2] = PR[GP1:90,2] + 14.089;
   1:L PR[91] R[100]mm/sec CNT100;
   1:  PR[GP1:91,1] = PR[GP1:90,1] + 62.657;
   1:  PR[GP1:91,2] = PR[GP1:90,2] + 18.812;
   1:L PR[91] R[100]mm/sec CNT100;
   1:  PR[GP1:91,1] = PR[GP1:90,1] + 58.919;
   1:  PR[GP1:91,2] = PR[GP1:90,2] + 23.649;
   1:L PR[91] R[100]mm/sec CNT100;
   1:  PR[GP1:91,1] = PR[GP1:90,1] + 58.489;
   1:  PR[GP1:91,2] = PR[GP1:90,2] + 24.103;
   1:L PR[91] R[100]mm/sec CNT100;
   1:  PR[GP1:91,1] = PR[GP1:90,1] + 53.872;
   1:  PR[GP1:91,2] = PR[GP1:90,2] + 28.230;
   1:L PR[91] R[100]mm/sec CNT100;
   1:  PR[GP1:91,1] = PR[GP1:90,1] + 53.666;
   1:  PR[GP1:91,2] = PR[GP1:90,2] + 28.396;
   1:L PR[91] R[100]mm/sec CNT100;
   1:  PR[GP1:91,1] = PR[GP1:90,1] + 48.047;
   1:  PR[GP1:91,2] = PR[GP1:90,2] + 31.879;
   1:L PR[91] R[100]mm/sec CNT100;
   1:  PR[GP1:91,1] = PR[GP1:90,1] + 42.517;
   1:  PR[GP1:91,2] = PR[GP1:90,2] + 34.088;
   1:L PR[91] R[100]mm/sec CNT100;
   1:  PR[GP1:91,1] = PR[GP1:90,1] + 40.755;
   1:  PR[GP1:91,2] = PR[GP1:90,2] + 34.710;
   1:L PR[91] R[100]mm/sec CNT100;
   1:  PR[GP1:91,1] = PR[GP1:90,1] + 35.039;
   1:  PR[GP1:91,2] = PR[GP1:90,2] + 35.940;
   1:L PR[91] R[100]mm/sec CNT100;
   1:  PR[GP1:91,1] = PR[GP1:90,1] + 29.882;
   1:  PR[GP1:91,2] = PR[GP1:90,2] + 36.135;
   1:L PR[91] R[100]mm/sec CNT100;
   1:  PR[GP1:91,1] = PR[GP1:90,1] + 26.365;
   1:  PR[GP1:91,2] = PR[GP1:90,2] + 36.147;
   1:L PR[91] R[100]mm/sec CNT100;
   1:  PR[GP1:91,1] = PR[GP1:90,1] + 21.419;
   1:  PR[GP1:91,2] = PR[GP1:90,2] + 35.497;
   1:L PR[91] R[100]mm/sec CNT100;
   1:  PR[GP1:91,1] = PR[GP1:90,1] + 17.177;
   1:  PR[GP1:91,2] = PR[GP1:90,2] + 34.147;
   1:L PR[91] R[100]mm/sec CNT100;
   1:  PR[GP1:91,1] = PR[GP1:90,1] + 12.531;
   1:  PR[GP1:91,2] = PR[GP1:90,2] + 32.536;
   1:L PR[91] R[100]mm/sec CNT100;
   1:  PR[GP1:91,1] = PR[GP1:90,1] + 8.825;
   1:  PR[GP1:91,2] = PR[GP1:90,2] + 30.602;
   1:L PR[91] R[100]mm/sec CNT100;
   1:  PR[GP1:91,1] = PR[GP1:90,1] + 6.533;
   1:  PR[GP1:91,2] = PR[GP1:90,2] + 28.983;
   1:L PR[91] R[100]mm/sec CNT100;
   1:  PR[GP1:91,1] = PR[GP1:90,1] + 4.885;
   1:  PR[GP1:91,2] = PR[GP1:90,2] + 27.694;
   1:L PR[91] R[100]mm/sec CNT100;
   1:  PR[GP1:91,1] = PR[GP1:90,1] + 3.566;
   1:  PR[GP1:91,2] = PR[GP1:90,2] + 26.158;
   1:L PR[91] R[100]mm/sec CNT100;
   1:  PR[GP1:91,1] = PR[GP1:90,1] + 2.069;
   1:  PR[GP1:91,2] = PR[GP1:90,2] + 25.567;
   1:L PR[91] R[100]mm/sec CNT100;
   1:  PR[GP1:91,1] = PR[GP1:90,1] + 1.125;
   1:  PR[GP1:91,2] = PR[GP1:90,2] + 25.084;
   1:L PR[91] R[100]mm/sec CNT100;
   1:  ! -- Layer/Ebene 85 -- !;
   1:  PR[91] = PR[90];
   1:  PR[GP1:91,1] = PR[GP1:90,1] + -2.099;
   1:  PR[GP1:91,2] = PR[GP1:90,2] + 25.834;
   1:  PR[GP1:91,3] = PR[GP1:90,3] + 52.155;
   1:L PR[91] R[100]mm/sec CNT100;
   1:  PR[GP1:91,1] = PR[GP1:90,1] + -3.343;
   1:  PR[GP1:91,2] = PR[GP1:90,2] + 26.467;
   1:L PR[91] R[100]mm/sec CNT100;
   1:  PR[GP1:91,1] = PR[GP1:90,1] + -4.504;
   1:  PR[GP1:91,2] = PR[GP1:90,2] + 27.817;
   1:L PR[91] R[100]mm/sec CNT100;
   1:  PR[GP1:91,1] = PR[GP1:90,1] + -5.987;
   1:  PR[GP1:91,2] = PR[GP1:90,2] + 28.979;
   1:L PR[91] R[100]mm/sec CNT100;
   1:  PR[GP1:91,1] = PR[GP1:90,1] + -8.392;
   1:  PR[GP1:91,2] = PR[GP1:90,2] + 30.678;
   1:L PR[91] R[100]mm/sec CNT100;
   1:  PR[GP1:91,1] = PR[GP1:90,1] + -11.984;
   1:  PR[GP1:91,2] = PR[GP1:90,2] + 32.557;
   1:L PR[91] R[100]mm/sec CNT100;
   1:  PR[GP1:91,1] = PR[GP1:90,1] + -16.398;
   1:  PR[GP1:91,2] = PR[GP1:90,2] + 33.975;
   1:L PR[91] R[100]mm/sec CNT100;
   1:  PR[GP1:91,1] = PR[GP1:90,1] + -21.020;
   1:  PR[GP1:91,2] = PR[GP1:90,2] + 35.573;
   1:L PR[91] R[100]mm/sec CNT100;
   1:  PR[GP1:91,1] = PR[GP1:90,1] + -25.803;
   1:  PR[GP1:91,2] = PR[GP1:90,2] + 36.198;
   1:L PR[91] R[100]mm/sec CNT100;
   1:  PR[GP1:91,1] = PR[GP1:90,1] + -31.401;
   1:  PR[GP1:91,2] = PR[GP1:90,2] + 36.006;
   1:L PR[91] R[100]mm/sec CNT100;
   1:  PR[GP1:91,1] = PR[GP1:90,1] + -34.684;
   1:  PR[GP1:91,2] = PR[GP1:90,2] + 35.989;
   1:L PR[91] R[100]mm/sec CNT100;
   1:  PR[GP1:91,1] = PR[GP1:90,1] + -40.230;
   1:  PR[GP1:91,2] = PR[GP1:90,2] + 34.793;
   1:L PR[91] R[100]mm/sec CNT100;
   1:  PR[GP1:91,1] = PR[GP1:90,1] + -46.293;
   1:  PR[GP1:91,2] = PR[GP1:90,2] + 32.392;
   1:L PR[91] R[100]mm/sec CNT100;
   1:  PR[GP1:91,1] = PR[GP1:90,1] + -47.693;
   1:  PR[GP1:91,2] = PR[GP1:90,2] + 31.895;
   1:L PR[91] R[100]mm/sec CNT100;
   1:  PR[GP1:91,1] = PR[GP1:90,1] + -53.183;
   1:  PR[GP1:91,2] = PR[GP1:90,2] + 28.475;
   1:L PR[91] R[100]mm/sec CNT100;
   1:  PR[GP1:91,1] = PR[GP1:90,1] + -58.440;
   1:  PR[GP1:91,2] = PR[GP1:90,2] + 23.795;
   1:L PR[91] R[100]mm/sec CNT100;
   1:  PR[GP1:91,1] = PR[GP1:90,1] + -62.350;
   1:  PR[GP1:91,2] = PR[GP1:90,2] + 18.721;
   1:L PR[91] R[100]mm/sec CNT100;
   1:  PR[GP1:91,1] = PR[GP1:90,1] + -65.669;
   1:  PR[GP1:91,2] = PR[GP1:90,2] + 12.133;
   1:L PR[91] R[100]mm/sec CNT100;
   1:  PR[GP1:91,1] = PR[GP1:90,1] + -67.137;
   1:  PR[GP1:91,2] = PR[GP1:90,2] + 7.148;
   1:L PR[91] R[100]mm/sec CNT100;
   1:  PR[GP1:91,1] = PR[GP1:90,1] + -67.480;
   1:  PR[GP1:91,2] = PR[GP1:90,2] + 4.948;
   1:L PR[91] R[100]mm/sec CNT100;
   1:  PR[GP1:91,1] = PR[GP1:90,1] + -67.929;
   1:  PR[GP1:91,2] = PR[GP1:90,2] + -0.052;
   1:L PR[91] R[100]mm/sec CNT100;
   1:  PR[GP1:91,1] = PR[GP1:90,1] + -67.575;
   1:  PR[GP1:91,2] = PR[GP1:90,2] + -2.296;
   1:L PR[91] R[100]mm/sec CNT100;
   1:  PR[GP1:91,1] = PR[GP1:90,1] + -67.131;
   1:  PR[GP1:91,2] = PR[GP1:90,2] + -7.311;
   1:L PR[91] R[100]mm/sec CNT100;
   1:  PR[GP1:91,1] = PR[GP1:90,1] + -65.669;
   1:  PR[GP1:91,2] = PR[GP1:90,2] + -12.277;
   1:L PR[91] R[100]mm/sec CNT100;
   1:  PR[GP1:91,1] = PR[GP1:90,1] + -62.350;
   1:  PR[GP1:91,2] = PR[GP1:90,2] + -18.865;
   1:L PR[91] R[100]mm/sec CNT100;
   1:  PR[GP1:91,1] = PR[GP1:90,1] + -58.439;
   1:  PR[GP1:91,2] = PR[GP1:90,2] + -23.940;
   1:L PR[91] R[100]mm/sec CNT100;
   1:  PR[GP1:91,1] = PR[GP1:90,1] + -53.650;
   1:  PR[GP1:91,2] = PR[GP1:90,2] + -28.245;
   1:L PR[91] R[100]mm/sec CNT100;
   1:  PR[GP1:91,1] = PR[GP1:90,1] + -53.195;
   1:  PR[GP1:91,2] = PR[GP1:90,2] + -28.612;
   1:L PR[91] R[100]mm/sec CNT100;
   1:  PR[GP1:91,1] = PR[GP1:90,1] + -47.681;
   1:  PR[GP1:91,2] = PR[GP1:90,2] + -32.046;
   1:L PR[91] R[100]mm/sec CNT100;
   1:  PR[GP1:91,1] = PR[GP1:90,1] + -42.296;
   1:  PR[GP1:91,2] = PR[GP1:90,2] + -34.209;
   1:L PR[91] R[100]mm/sec CNT100;
   1:  PR[GP1:91,1] = PR[GP1:90,1] + -40.238;
   1:  PR[GP1:91,2] = PR[GP1:90,2] + -34.935;
   1:L PR[91] R[100]mm/sec CNT100;
   1:  PR[GP1:91,1] = PR[GP1:90,1] + -34.670;
   1:  PR[GP1:91,2] = PR[GP1:90,2] + -36.136;
   1:L PR[91] R[100]mm/sec CNT100;
   1:  PR[GP1:91,1] = PR[GP1:90,1] + -29.630;
   1:  PR[GP1:91,2] = PR[GP1:90,2] + -36.330;
   1:L PR[91] R[100]mm/sec CNT100;
   1:  PR[GP1:91,1] = PR[GP1:90,1] + -25.806;
   1:  PR[GP1:91,2] = PR[GP1:90,2] + -36.342;
   1:L PR[91] R[100]mm/sec CNT100;
   1:  PR[GP1:91,1] = PR[GP1:90,1] + -21.005;
   1:  PR[GP1:91,2] = PR[GP1:90,2] + -35.715;
   1:L PR[91] R[100]mm/sec CNT100;
   1:  PR[GP1:91,1] = PR[GP1:90,1] + -16.899;
   1:  PR[GP1:91,2] = PR[GP1:90,2] + -34.408;
   1:L PR[91] R[100]mm/sec CNT100;
   1:  PR[GP1:91,1] = PR[GP1:90,1] + -11.982;
   1:  PR[GP1:91,2] = PR[GP1:90,2] + -32.700;
   1:L PR[91] R[100]mm/sec CNT100;
   1:  PR[GP1:91,1] = PR[GP1:90,1] + -8.390;
   1:  PR[GP1:91,2] = PR[GP1:90,2] + -30.820;
   1:L PR[91] R[100]mm/sec CNT100;
   1:  PR[GP1:91,1] = PR[GP1:90,1] + -5.070;
   1:  PR[GP1:91,2] = PR[GP1:90,2] + -28.408;
   1:L PR[91] R[100]mm/sec CNT100;
   1:  PR[GP1:91,1] = PR[GP1:90,1] + -4.107;
   1:  PR[GP1:91,2] = PR[GP1:90,2] + -27.655;
   1:L PR[91] R[100]mm/sec CNT100;
   1:  PR[GP1:91,1] = PR[GP1:90,1] + -3.286;
   1:  PR[GP1:91,2] = PR[GP1:90,2] + -26.701;
   1:L PR[91] R[100]mm/sec CNT100;
   1:  PR[GP1:91,1] = PR[GP1:90,1] + 0.202;
   1:  PR[GP1:91,2] = PR[GP1:90,2] + -25.953;
   1:L PR[91] R[100]mm/sec CNT100;
   1:  PR[GP1:91,1] = PR[GP1:90,1] + 1.052;
   1:  PR[GP1:91,2] = PR[GP1:90,2] + -25.502;
   1:L PR[91] R[100]mm/sec CNT100;
   1:  PR[GP1:91,1] = PR[GP1:90,1] + 3.552;
   1:  PR[GP1:91,2] = PR[GP1:90,2] + -26.765;
   1:L PR[91] R[100]mm/sec CNT100;
   1:  PR[GP1:91,1] = PR[GP1:90,1] + 4.327;
   1:  PR[GP1:91,2] = PR[GP1:90,2] + -27.665;
   1:L PR[91] R[100]mm/sec CNT100;
   1:  PR[GP1:91,1] = PR[GP1:90,1] + 5.285;
   1:  PR[GP1:91,2] = PR[GP1:90,2] + -28.414;
   1:L PR[91] R[100]mm/sec CNT100;
   1:  PR[GP1:91,1] = PR[GP1:90,1] + 8.612;
   1:  PR[GP1:91,2] = PR[GP1:90,2] + -30.832;
   1:L PR[91] R[100]mm/sec CNT100;
   1:  PR[GP1:91,1] = PR[GP1:90,1] + 12.175;
   1:  PR[GP1:91,2] = PR[GP1:90,2] + -32.691;
   1:L PR[91] R[100]mm/sec CNT100;
   1:  PR[GP1:91,1] = PR[GP1:90,1] + 16.593;
   1:  PR[GP1:91,2] = PR[GP1:90,2] + -34.110;
   1:L PR[91] R[100]mm/sec CNT100;
   1:  PR[GP1:91,1] = PR[GP1:90,1] + 21.221;
   1:  PR[GP1:91,2] = PR[GP1:90,2] + -35.713;
   1:L PR[91] R[100]mm/sec CNT100;
   1:  PR[GP1:91,1] = PR[GP1:90,1] + 25.998;
   1:  PR[GP1:91,2] = PR[GP1:90,2] + -36.341;
   1:L PR[91] R[100]mm/sec CNT100;
   1:  PR[GP1:91,1] = PR[GP1:90,1] + 31.570;
   1:  PR[GP1:91,2] = PR[GP1:90,2] + -36.154;
   1:L PR[91] R[100]mm/sec CNT100;
   1:  PR[GP1:91,1] = PR[GP1:90,1] + 34.859;
   1:  PR[GP1:91,2] = PR[GP1:90,2] + -36.139;
   1:L PR[91] R[100]mm/sec CNT100;
   1:  PR[GP1:91,1] = PR[GP1:90,1] + 40.397;
   1:  PR[GP1:91,2] = PR[GP1:90,2] + -34.947;
   1:L PR[91] R[100]mm/sec CNT100;
   1:  PR[GP1:91,1] = PR[GP1:90,1] + 46.469;
   1:  PR[GP1:91,2] = PR[GP1:90,2] + -32.555;
   1:L PR[91] R[100]mm/sec CNT100;
   1:  PR[GP1:91,1] = PR[GP1:90,1] + 47.873;
   1:  PR[GP1:91,2] = PR[GP1:90,2] + -32.057;
   1:L PR[91] R[100]mm/sec CNT100;
   1:  PR[GP1:91,1] = PR[GP1:90,1] + 53.330;
   1:  PR[GP1:91,2] = PR[GP1:90,2] + -28.675;
   1:L PR[91] R[100]mm/sec CNT100;
   1:  PR[GP1:91,1] = PR[GP1:90,1] + 58.562;
   1:  PR[GP1:91,2] = PR[GP1:90,2] + -24.032;
   1:L PR[91] R[100]mm/sec CNT100;
   1:  PR[GP1:91,1] = PR[GP1:90,1] + 62.530;
   1:  PR[GP1:91,2] = PR[GP1:90,2] + -18.898;
   1:L PR[91] R[100]mm/sec CNT100;
   1:  PR[GP1:91,1] = PR[GP1:90,1] + 65.860;
   1:  PR[GP1:91,2] = PR[GP1:90,2] + -12.356;
   1:L PR[91] R[100]mm/sec CNT100;
   1:  PR[GP1:91,1] = PR[GP1:90,1] + 67.328;
   1:  PR[GP1:91,2] = PR[GP1:90,2] + -7.437;
   1:L PR[91] R[100]mm/sec CNT100;
   1:  PR[GP1:91,1] = PR[GP1:90,1] + 67.670;
   1:  PR[GP1:91,2] = PR[GP1:90,2] + -5.235;
   1:L PR[91] R[100]mm/sec CNT100;
   1:  PR[GP1:91,1] = PR[GP1:90,1] + 68.142;
   1:  PR[GP1:91,2] = PR[GP1:90,2] + -0.092;
   1:L PR[91] R[100]mm/sec CNT100;
   1:  PR[GP1:91,1] = PR[GP1:90,1] + 67.788;
   1:  PR[GP1:91,2] = PR[GP1:90,2] + 2.158;
   1:L PR[91] R[100]mm/sec CNT100;
   1:  PR[GP1:91,1] = PR[GP1:90,1] + 67.322;
   1:  PR[GP1:91,2] = PR[GP1:90,2] + 7.312;
   1:L PR[91] R[100]mm/sec CNT100;
   1:  PR[GP1:91,1] = PR[GP1:90,1] + 65.860;
   1:  PR[GP1:91,2] = PR[GP1:90,2] + 12.212;
   1:L PR[91] R[100]mm/sec CNT100;
   1:  PR[GP1:91,1] = PR[GP1:90,1] + 62.530;
   1:  PR[GP1:91,2] = PR[GP1:90,2] + 18.754;
   1:L PR[91] R[100]mm/sec CNT100;
   1:  PR[GP1:91,1] = PR[GP1:90,1] + 58.518;
   1:  PR[GP1:91,2] = PR[GP1:90,2] + 23.936;
   1:L PR[91] R[100]mm/sec CNT100;
   1:  PR[GP1:91,1] = PR[GP1:90,1] + 53.803;
   1:  PR[GP1:91,2] = PR[GP1:90,2] + 28.151;
   1:L PR[91] R[100]mm/sec CNT100;
   1:  PR[GP1:91,1] = PR[GP1:90,1] + 53.343;
   1:  PR[GP1:91,2] = PR[GP1:90,2] + 28.523;
   1:L PR[91] R[100]mm/sec CNT100;
   1:  PR[GP1:91,1] = PR[GP1:90,1] + 47.864;
   1:  PR[GP1:91,2] = PR[GP1:90,2] + 31.919;
   1:L PR[91] R[100]mm/sec CNT100;
   1:  PR[GP1:91,1] = PR[GP1:90,1] + 42.472;
   1:  PR[GP1:91,2] = PR[GP1:90,2] + 34.073;
   1:L PR[91] R[100]mm/sec CNT100;
   1:  PR[GP1:91,1] = PR[GP1:90,1] + 40.410;
   1:  PR[GP1:91,2] = PR[GP1:90,2] + 34.800;
   1:L PR[91] R[100]mm/sec CNT100;
   1:  PR[GP1:91,1] = PR[GP1:90,1] + 34.853;
   1:  PR[GP1:91,2] = PR[GP1:90,2] + 35.997;
   1:L PR[91] R[100]mm/sec CNT100;
   1:  PR[GP1:91,1] = PR[GP1:90,1] + 29.837;
   1:  PR[GP1:91,2] = PR[GP1:90,2] + 36.186;
   1:L PR[91] R[100]mm/sec CNT100;
   1:  PR[GP1:91,1] = PR[GP1:90,1] + 26.013;
   1:  PR[GP1:91,2] = PR[GP1:90,2] + 36.199;
   1:L PR[91] R[100]mm/sec CNT100;
   1:  PR[GP1:91,1] = PR[GP1:90,1] + 21.221;
   1:  PR[GP1:91,2] = PR[GP1:90,2] + 35.569;
   1:L PR[91] R[100]mm/sec CNT100;
   1:  PR[GP1:91,1] = PR[GP1:90,1] + 17.109;
   1:  PR[GP1:91,2] = PR[GP1:90,2] + 34.261;
   1:L PR[91] R[100]mm/sec CNT100;
   1:  PR[GP1:91,1] = PR[GP1:90,1] + 12.190;
   1:  PR[GP1:91,2] = PR[GP1:90,2] + 32.555;
   1:L PR[91] R[100]mm/sec CNT100;
   1:  PR[GP1:91,1] = PR[GP1:90,1] + 8.614;
   1:  PR[GP1:91,2] = PR[GP1:90,2] + 30.689;
   1:L PR[91] R[100]mm/sec CNT100;
   1:  PR[GP1:91,1] = PR[GP1:90,1] + 6.203;
   1:  PR[GP1:91,2] = PR[GP1:90,2] + 28.986;
   1:L PR[91] R[100]mm/sec CNT100;
   1:  PR[GP1:91,1] = PR[GP1:90,1] + 4.728;
   1:  PR[GP1:91,2] = PR[GP1:90,2] + 27.832;
   1:L PR[91] R[100]mm/sec CNT100;
   1:  PR[GP1:91,1] = PR[GP1:90,1] + 3.536;
   1:  PR[GP1:91,2] = PR[GP1:90,2] + 26.445;
   1:L PR[91] R[100]mm/sec CNT100;
   1:  PR[GP1:91,1] = PR[GP1:90,1] + 1.980;
   1:  PR[GP1:91,2] = PR[GP1:90,2] + 25.830;
   1:L PR[91] R[100]mm/sec CNT100;
   1:  PR[GP1:91,1] = PR[GP1:90,1] + 1.166;
   1:  PR[GP1:91,2] = PR[GP1:90,2] + 25.414;
   1:L PR[91] R[100]mm/sec CNT100;
   1:  ! -- Layer/Ebene 86 -- !;
   1:  PR[91] = PR[90];
   1:  PR[GP1:91,1] = PR[GP1:90,1] + -2.187;
   1:  PR[GP1:91,2] = PR[GP1:90,2] + 26.180;
   1:  PR[GP1:91,3] = PR[GP1:90,3] + 52.765;
   1:L PR[91] R[100]mm/sec CNT100;
   1:  PR[GP1:91,1] = PR[GP1:90,1] + -3.313;
   1:  PR[GP1:91,2] = PR[GP1:90,2] + 26.753;
   1:L PR[91] R[100]mm/sec CNT100;
   1:  PR[GP1:91,1] = PR[GP1:90,1] + -4.349;
   1:  PR[GP1:91,2] = PR[GP1:90,2] + 27.957;
   1:L PR[91] R[100]mm/sec CNT100;
   1:  PR[GP1:91,1] = PR[GP1:90,1] + -5.657;
   1:  PR[GP1:91,2] = PR[GP1:90,2] + 28.982;
   1:L PR[91] R[100]mm/sec CNT100;
   1:  PR[GP1:91,1] = PR[GP1:90,1] + -8.181;
   1:  PR[GP1:91,2] = PR[GP1:90,2] + 30.765;
   1:L PR[91] R[100]mm/sec CNT100;
   1:  PR[GP1:91,1] = PR[GP1:90,1] + -11.642;
   1:  PR[GP1:91,2] = PR[GP1:90,2] + 32.576;
   1:L PR[91] R[100]mm/sec CNT100;
   1:  PR[GP1:91,1] = PR[GP1:90,1] + -15.897;
   1:  PR[GP1:91,2] = PR[GP1:90,2] + 33.943;
   1:L PR[91] R[100]mm/sec CNT100;
   1:  PR[GP1:91,1] = PR[GP1:90,1] + -20.822;
   1:  PR[GP1:91,2] = PR[GP1:90,2] + 35.645;
   1:L PR[91] R[100]mm/sec CNT100;
   1:  PR[GP1:91,1] = PR[GP1:90,1] + -25.451;
   1:  PR[GP1:91,2] = PR[GP1:90,2] + 36.250;
   1:L PR[91] R[100]mm/sec CNT100;
   1:  PR[GP1:91,1] = PR[GP1:90,1] + -30.873;
   1:  PR[GP1:91,2] = PR[GP1:90,2] + 36.064;
   1:L PR[91] R[100]mm/sec CNT100;
   1:  PR[GP1:91,1] = PR[GP1:90,1] + -34.496;
   1:  PR[GP1:91,2] = PR[GP1:90,2] + 36.046;
   1:L PR[91] R[100]mm/sec CNT100;
   1:  PR[GP1:91,1] = PR[GP1:90,1] + -39.884;
   1:  PR[GP1:91,2] = PR[GP1:90,2] + 34.884;
   1:L PR[91] R[100]mm/sec CNT100;
   1:  PR[GP1:91,1] = PR[GP1:90,1] + -45.777;
   1:  PR[GP1:91,2] = PR[GP1:90,2] + 32.550;
   1:L PR[91] R[100]mm/sec CNT100;
   1:  PR[GP1:91,1] = PR[GP1:90,1] + -47.509;
   1:  PR[GP1:91,2] = PR[GP1:90,2] + 31.935;
   1:L PR[91] R[100]mm/sec CNT100;
   1:  PR[GP1:91,1] = PR[GP1:90,1] + -52.859;
   1:  PR[GP1:91,2] = PR[GP1:90,2] + 28.603;
   1:L PR[91] R[100]mm/sec CNT100;
   1:  PR[GP1:91,1] = PR[GP1:90,1] + -58.046;
   1:  PR[GP1:91,2] = PR[GP1:90,2] + 23.997;
   1:L PR[91] R[100]mm/sec CNT100;
   1:  PR[GP1:91,1] = PR[GP1:90,1] + -58.240;
   1:  PR[GP1:91,2] = PR[GP1:90,2] + 23.840;
   1:L PR[91] R[100]mm/sec CNT100;
   1:  PR[GP1:91,1] = PR[GP1:90,1] + -62.225;
   1:  PR[GP1:91,2] = PR[GP1:90,2] + 18.660;
   1:L PR[91] R[100]mm/sec CNT100;
   1:  PR[GP1:91,1] = PR[GP1:90,1] + -65.453;
   1:  PR[GP1:91,2] = PR[GP1:90,2] + 12.259;
   1:L PR[91] R[100]mm/sec CNT100;
   1:  PR[GP1:91,1] = PR[GP1:90,1] + -67.020;
   1:  PR[GP1:91,2] = PR[GP1:90,2] + 6.934;
   1:L PR[91] R[100]mm/sec CNT100;
   1:  PR[GP1:91,1] = PR[GP1:90,1] + -67.273;
   1:  PR[GP1:91,2] = PR[GP1:90,2] + 5.311;
   1:L PR[91] R[100]mm/sec CNT100;
   1:  PR[GP1:91,1] = PR[GP1:90,1] + -67.755;
   1:  PR[GP1:91,2] = PR[GP1:90,2] + -0.052;
   1:L PR[91] R[100]mm/sec CNT100;
   1:  PR[GP1:91,1] = PR[GP1:90,1] + -67.488;
   1:  PR[GP1:91,2] = PR[GP1:90,2] + -1.743;
   1:L PR[91] R[100]mm/sec CNT100;
   1:  PR[GP1:91,1] = PR[GP1:90,1] + -67.015;
   1:  PR[GP1:91,2] = PR[GP1:90,2] + -7.097;
   1:L PR[91] R[100]mm/sec CNT100;
   1:  PR[GP1:91,1] = PR[GP1:90,1] + -65.453;
   1:  PR[GP1:91,2] = PR[GP1:90,2] + -12.403;
   1:L PR[91] R[100]mm/sec CNT100;
   1:  PR[GP1:91,1] = PR[GP1:90,1] + -62.225;
   1:  PR[GP1:91,2] = PR[GP1:90,2] + -18.804;
   1:L PR[91] R[100]mm/sec CNT100;
   1:  PR[GP1:91,1] = PR[GP1:90,1] + -58.230;
   1:  PR[GP1:91,2] = PR[GP1:90,2] + -23.996;
   1:L PR[91] R[100]mm/sec CNT100;
   1:  PR[GP1:91,1] = PR[GP1:90,1] + -53.580;
   1:  PR[GP1:91,2] = PR[GP1:90,2] + -28.168;
   1:L PR[91] R[100]mm/sec CNT100;
   1:  PR[GP1:91,1] = PR[GP1:90,1] + -52.870;
   1:  PR[GP1:91,2] = PR[GP1:90,2] + -28.740;
   1:L PR[91] R[100]mm/sec CNT100;
   1:  PR[GP1:91,1] = PR[GP1:90,1] + -47.497;
   1:  PR[GP1:91,2] = PR[GP1:90,2] + -32.087;
   1:L PR[91] R[100]mm/sec CNT100;
   1:  PR[GP1:91,1] = PR[GP1:90,1] + -42.250;
   1:  PR[GP1:91,2] = PR[GP1:90,2] + -34.194;
   1:L PR[91] R[100]mm/sec CNT100;
   1:  PR[GP1:91,1] = PR[GP1:90,1] + -39.892;
   1:  PR[GP1:91,2] = PR[GP1:90,2] + -35.026;
   1:L PR[91] R[100]mm/sec CNT100;
   1:  PR[GP1:91,1] = PR[GP1:90,1] + -34.482;
   1:  PR[GP1:91,2] = PR[GP1:90,2] + -36.193;
   1:L PR[91] R[100]mm/sec CNT100;
   1:  PR[GP1:91,1] = PR[GP1:90,1] + -29.584;
   1:  PR[GP1:91,2] = PR[GP1:90,2] + -36.381;
   1:L PR[91] R[100]mm/sec CNT100;
   1:  PR[GP1:91,1] = PR[GP1:90,1] + -25.454;
   1:  PR[GP1:91,2] = PR[GP1:90,2] + -36.394;
   1:L PR[91] R[100]mm/sec CNT100;
   1:  PR[GP1:91,1] = PR[GP1:90,1] + -20.806;
   1:  PR[GP1:91,2] = PR[GP1:90,2] + -35.787;
   1:L PR[91] R[100]mm/sec CNT100;
   1:  PR[GP1:91,1] = PR[GP1:90,1] + -16.830;
   1:  PR[GP1:91,2] = PR[GP1:90,2] + -34.522;
   1:L PR[91] R[100]mm/sec CNT100;
   1:  PR[GP1:91,1] = PR[GP1:90,1] + -11.640;
   1:  PR[GP1:91,2] = PR[GP1:90,2] + -32.718;
   1:L PR[91] R[100]mm/sec CNT100;
   1:  PR[GP1:91,1] = PR[GP1:90,1] + -8.179;
   1:  PR[GP1:91,2] = PR[GP1:90,2] + -30.908;
   1:L PR[91] R[100]mm/sec CNT100;
   1:  PR[GP1:91,1] = PR[GP1:90,1] + -4.696;
   1:  PR[GP1:91,2] = PR[GP1:90,2] + -28.377;
   1:L PR[91] R[100]mm/sec CNT100;
   1:  PR[GP1:91,1] = PR[GP1:90,1] + -3.934;
   1:  PR[GP1:91,2] = PR[GP1:90,2] + -27.780;
   1:L PR[91] R[100]mm/sec CNT100;
   1:  PR[GP1:91,1] = PR[GP1:90,1] + -3.256;
   1:  PR[GP1:91,2] = PR[GP1:90,2] + -26.994;
   1:L PR[91] R[100]mm/sec CNT100;
   1:  PR[GP1:91,1] = PR[GP1:90,1] + 0.369;
   1:  PR[GP1:91,2] = PR[GP1:90,2] + -26.216;
   1:L PR[91] R[100]mm/sec CNT100;
   1:  PR[GP1:91,1] = PR[GP1:90,1] + 1.093;
   1:  PR[GP1:91,2] = PR[GP1:90,2] + -25.832;
   1:L PR[91] R[100]mm/sec CNT100;
   1:  PR[GP1:91,1] = PR[GP1:90,1] + 3.522;
   1:  PR[GP1:91,2] = PR[GP1:90,2] + -27.058;
   1:L PR[91] R[100]mm/sec CNT100;
   1:  PR[GP1:91,1] = PR[GP1:90,1] + 4.152;
   1:  PR[GP1:91,2] = PR[GP1:90,2] + -27.789;
   1:L PR[91] R[100]mm/sec CNT100;
   1:  PR[GP1:91,1] = PR[GP1:90,1] + 4.909;
   1:  PR[GP1:91,2] = PR[GP1:90,2] + -28.382;
   1:L PR[91] R[100]mm/sec CNT100;
   1:  PR[GP1:91,1] = PR[GP1:90,1] + 8.401;
   1:  PR[GP1:91,2] = PR[GP1:90,2] + -30.918;
   1:L PR[91] R[100]mm/sec CNT100;
   1:  PR[GP1:91,1] = PR[GP1:90,1] + 11.833;
   1:  PR[GP1:91,2] = PR[GP1:90,2] + -32.710;
   1:L PR[91] R[100]mm/sec CNT100;
   1:  PR[GP1:91,1] = PR[GP1:90,1] + 16.091;
   1:  PR[GP1:91,2] = PR[GP1:90,2] + -34.078;
   1:L PR[91] R[100]mm/sec CNT100;
   1:  PR[GP1:91,1] = PR[GP1:90,1] + 21.023;
   1:  PR[GP1:91,2] = PR[GP1:90,2] + -35.785;
   1:L PR[91] R[100]mm/sec CNT100;
   1:  PR[GP1:91,1] = PR[GP1:90,1] + 25.646;
   1:  PR[GP1:91,2] = PR[GP1:90,2] + -36.393;
   1:L PR[91] R[100]mm/sec CNT100;
   1:  PR[GP1:91,1] = PR[GP1:90,1] + 31.042;
   1:  PR[GP1:91,2] = PR[GP1:90,2] + -36.212;
   1:L PR[91] R[100]mm/sec CNT100;
   1:  PR[GP1:91,1] = PR[GP1:90,1] + 34.671;
   1:  PR[GP1:91,2] = PR[GP1:90,2] + -36.196;
   1:L PR[91] R[100]mm/sec CNT100;
   1:  PR[GP1:91,1] = PR[GP1:90,1] + 40.052;
   1:  PR[GP1:91,2] = PR[GP1:90,2] + -35.038;
   1:L PR[91] R[100]mm/sec CNT100;
   1:  PR[GP1:91,1] = PR[GP1:90,1] + 45.953;
   1:  PR[GP1:91,2] = PR[GP1:90,2] + -32.713;
   1:L PR[91] R[100]mm/sec CNT100;
   1:  PR[GP1:91,1] = PR[GP1:90,1] + 47.690;
   1:  PR[GP1:91,2] = PR[GP1:90,2] + -32.097;
   1:L PR[91] R[100]mm/sec CNT100;
   1:  PR[GP1:91,1] = PR[GP1:90,1] + 53.007;
   1:  PR[GP1:91,2] = PR[GP1:90,2] + -28.802;
   1:L PR[91] R[100]mm/sec CNT100;
   1:  PR[GP1:91,1] = PR[GP1:90,1] + 58.166;
   1:  PR[GP1:91,2] = PR[GP1:90,2] + -24.234;
   1:L PR[91] R[100]mm/sec CNT100;
   1:  PR[GP1:91,1] = PR[GP1:90,1] + 58.369;
   1:  PR[GP1:91,2] = PR[GP1:90,2] + -24.069;
   1:L PR[91] R[100]mm/sec CNT100;
   1:  PR[GP1:91,1] = PR[GP1:90,1] + 62.403;
   1:  PR[GP1:91,2] = PR[GP1:90,2] + -18.840;
   1:L PR[91] R[100]mm/sec CNT100;
   1:  PR[GP1:91,1] = PR[GP1:90,1] + 65.642;
   1:  PR[GP1:91,2] = PR[GP1:90,2] + -12.486;
   1:L PR[91] R[100]mm/sec CNT100;
   1:  PR[GP1:91,1] = PR[GP1:90,1] + 67.210;
   1:  PR[GP1:91,2] = PR[GP1:90,2] + -7.231;
   1:L PR[91] R[100]mm/sec CNT100;
   1:  PR[GP1:91,1] = PR[GP1:90,1] + 67.462;
   1:  PR[GP1:91,2] = PR[GP1:90,2] + -5.609;
   1:L PR[91] R[100]mm/sec CNT100;
   1:  PR[GP1:91,1] = PR[GP1:90,1] + 67.969;
   1:  PR[GP1:91,2] = PR[GP1:90,2] + -0.092;
   1:L PR[91] R[100]mm/sec CNT100;
   1:  PR[GP1:91,1] = PR[GP1:90,1] + 67.702;
   1:  PR[GP1:91,2] = PR[GP1:90,2] + 1.603;
   1:L PR[91] R[100]mm/sec CNT100;
   1:  PR[GP1:91,1] = PR[GP1:90,1] + 67.204;
   1:  PR[GP1:91,2] = PR[GP1:90,2] + 7.106;
   1:L PR[91] R[100]mm/sec CNT100;
   1:  PR[GP1:91,1] = PR[GP1:90,1] + 65.642;
   1:  PR[GP1:91,2] = PR[GP1:90,2] + 12.342;
   1:L PR[91] R[100]mm/sec CNT100;
   1:  PR[GP1:91,1] = PR[GP1:90,1] + 62.403;
   1:  PR[GP1:91,2] = PR[GP1:90,2] + 18.696;
   1:L PR[91] R[100]mm/sec CNT100;
   1:  PR[GP1:91,1] = PR[GP1:90,1] + 58.360;
   1:  PR[GP1:91,2] = PR[GP1:90,2] + 23.936;
   1:L PR[91] R[100]mm/sec CNT100;
   1:  PR[GP1:91,1] = PR[GP1:90,1] + 53.735;
   1:  PR[GP1:91,2] = PR[GP1:90,2] + 28.072;
   1:L PR[91] R[100]mm/sec CNT100;
   1:  PR[GP1:91,1] = PR[GP1:90,1] + 53.020;
   1:  PR[GP1:91,2] = PR[GP1:90,2] + 28.650;
   1:L PR[91] R[100]mm/sec CNT100;
   1:  PR[GP1:91,1] = PR[GP1:90,1] + 47.682;
   1:  PR[GP1:91,2] = PR[GP1:90,2] + 31.959;
   1:L PR[91] R[100]mm/sec CNT100;
   1:  PR[GP1:91,1] = PR[GP1:90,1] + 42.427;
   1:  PR[GP1:91,2] = PR[GP1:90,2] + 34.057;
   1:L PR[91] R[100]mm/sec CNT100;
   1:  PR[GP1:91,1] = PR[GP1:90,1] + 40.066;
   1:  PR[GP1:91,2] = PR[GP1:90,2] + 34.891;
   1:L PR[91] R[100]mm/sec CNT100;
   1:  PR[GP1:91,1] = PR[GP1:90,1] + 34.666;
   1:  PR[GP1:91,2] = PR[GP1:90,2] + 36.053;
   1:L PR[91] R[100]mm/sec CNT100;
   1:  PR[GP1:91,1] = PR[GP1:90,1] + 29.792;
   1:  PR[GP1:91,2] = PR[GP1:90,2] + 36.237;
   1:L PR[91] R[100]mm/sec CNT100;
   1:  PR[GP1:91,1] = PR[GP1:90,1] + 25.662;
   1:  PR[GP1:91,2] = PR[GP1:90,2] + 36.251;
   1:L PR[91] R[100]mm/sec CNT100;
   1:  PR[GP1:91,1] = PR[GP1:90,1] + 21.023;
   1:  PR[GP1:91,2] = PR[GP1:90,2] + 35.641;
   1:L PR[91] R[100]mm/sec CNT100;
   1:  PR[GP1:91,1] = PR[GP1:90,1] + 17.042;
   1:  PR[GP1:91,2] = PR[GP1:90,2] + 34.375;
   1:L PR[91] R[100]mm/sec CNT100;
   1:  PR[GP1:91,1] = PR[GP1:90,1] + 11.848;
   1:  PR[GP1:91,2] = PR[GP1:90,2] + 32.574;
   1:L PR[91] R[100]mm/sec CNT100;
   1:  PR[GP1:91,1] = PR[GP1:90,1] + 8.402;
   1:  PR[GP1:91,2] = PR[GP1:90,2] + 30.776;
   1:L PR[91] R[100]mm/sec CNT100;
   1:  PR[GP1:91,1] = PR[GP1:90,1] + 5.872;
   1:  PR[GP1:91,2] = PR[GP1:90,2] + 28.989;
   1:L PR[91] R[100]mm/sec CNT100;
   1:  PR[GP1:91,1] = PR[GP1:90,1] + 4.570;
   1:  PR[GP1:91,2] = PR[GP1:90,2] + 27.970;
   1:L PR[91] R[100]mm/sec CNT100;
   1:  PR[GP1:91,1] = PR[GP1:90,1] + 3.506;
   1:  PR[GP1:91,2] = PR[GP1:90,2] + 26.731;
   1:L PR[91] R[100]mm/sec CNT100;
   1:  PR[GP1:91,1] = PR[GP1:90,1] + 1.891;
   1:  PR[GP1:91,2] = PR[GP1:90,2] + 26.094;
   1:L PR[91] R[100]mm/sec CNT100;
   1:  PR[GP1:91,1] = PR[GP1:90,1] + 1.207;
   1:  PR[GP1:91,2] = PR[GP1:90,2] + 25.744;
   1:L PR[91] R[100]mm/sec CNT100;
   1:  ! -- Layer/Ebene 87 -- !;
   1:  PR[91] = PR[90];
   1:  PR[GP1:91,1] = PR[GP1:90,1] + -2.276;
   1:  PR[GP1:91,2] = PR[GP1:90,2] + 26.527;
   1:  PR[GP1:91,3] = PR[GP1:90,3] + 53.375;
   1:L PR[91] R[100]mm/sec CNT100;
   1:  PR[GP1:91,1] = PR[GP1:90,1] + -3.284;
   1:  PR[GP1:91,2] = PR[GP1:90,2] + 27.040;
   1:L PR[91] R[100]mm/sec CNT100;
   1:  PR[GP1:91,1] = PR[GP1:90,1] + -4.193;
   1:  PR[GP1:91,2] = PR[GP1:90,2] + 28.096;
   1:L PR[91] R[100]mm/sec CNT100;
   1:  PR[GP1:91,1] = PR[GP1:90,1] + -5.328;
   1:  PR[GP1:91,2] = PR[GP1:90,2] + 28.985;
   1:L PR[91] R[100]mm/sec CNT100;
   1:  PR[GP1:91,1] = PR[GP1:90,1] + -7.970;
   1:  PR[GP1:91,2] = PR[GP1:90,2] + 30.852;
   1:L PR[91] R[100]mm/sec CNT100;
   1:  PR[GP1:91,1] = PR[GP1:90,1] + -11.300;
   1:  PR[GP1:91,2] = PR[GP1:90,2] + 32.595;
   1:L PR[91] R[100]mm/sec CNT100;
   1:  PR[GP1:91,1] = PR[GP1:90,1] + -15.396;
   1:  PR[GP1:91,2] = PR[GP1:90,2] + 33.911;
   1:L PR[91] R[100]mm/sec CNT100;
   1:  PR[GP1:91,1] = PR[GP1:90,1] + -20.623;
   1:  PR[GP1:91,2] = PR[GP1:90,2] + 35.718;
   1:L PR[91] R[100]mm/sec CNT100;
   1:  PR[GP1:91,1] = PR[GP1:90,1] + -25.100;
   1:  PR[GP1:91,2] = PR[GP1:90,2] + 36.303;
   1:L PR[91] R[100]mm/sec CNT100;
   1:  PR[GP1:91,1] = PR[GP1:90,1] + -30.345;
   1:  PR[GP1:91,2] = PR[GP1:90,2] + 36.122;
   1:L PR[91] R[100]mm/sec CNT100;
   1:  PR[GP1:91,1] = PR[GP1:90,1] + -34.308;
   1:  PR[GP1:91,2] = PR[GP1:90,2] + 36.102;
   1:L PR[91] R[100]mm/sec CNT100;
   1:  PR[GP1:91,1] = PR[GP1:90,1] + -39.539;
   1:  PR[GP1:91,2] = PR[GP1:90,2] + 34.974;
   1:L PR[91] R[100]mm/sec CNT100;
   1:  PR[GP1:91,1] = PR[GP1:90,1] + -45.262;
   1:  PR[GP1:91,2] = PR[GP1:90,2] + 32.708;
   1:L PR[91] R[100]mm/sec CNT100;
   1:  PR[GP1:91,1] = PR[GP1:90,1] + -47.326;
   1:  PR[GP1:91,2] = PR[GP1:90,2] + 31.975;
   1:L PR[91] R[100]mm/sec CNT100;
   1:  PR[GP1:91,1] = PR[GP1:90,1] + -52.534;
   1:  PR[GP1:91,2] = PR[GP1:90,2] + 28.731;
   1:L PR[91] R[100]mm/sec CNT100;
   1:  PR[GP1:91,1] = PR[GP1:90,1] + -57.585;
   1:  PR[GP1:91,2] = PR[GP1:90,2] + 24.245;
   1:L PR[91] R[100]mm/sec CNT100;
   1:  PR[GP1:91,1] = PR[GP1:90,1] + -58.056;
   1:  PR[GP1:91,2] = PR[GP1:90,2] + 23.864;
   1:L PR[91] R[100]mm/sec CNT100;
   1:  PR[GP1:91,1] = PR[GP1:90,1] + -62.075;
   1:  PR[GP1:91,2] = PR[GP1:90,2] + 18.633;
   1:L PR[91] R[100]mm/sec CNT100;
   1:  PR[GP1:91,1] = PR[GP1:90,1] + -65.236;
   1:  PR[GP1:91,2] = PR[GP1:90,2] + 12.385;
   1:L PR[91] R[100]mm/sec CNT100;
   1:  PR[GP1:91,1] = PR[GP1:90,1] + -66.904;
   1:  PR[GP1:91,2] = PR[GP1:90,2] + 6.720;
   1:L PR[91] R[100]mm/sec CNT100;
   1:  PR[GP1:91,1] = PR[GP1:90,1] + -67.067;
   1:  PR[GP1:91,2] = PR[GP1:90,2] + 5.675;
   1:L PR[91] R[100]mm/sec CNT100;
   1:  PR[GP1:91,1] = PR[GP1:90,1] + -67.581;
   1:  PR[GP1:91,2] = PR[GP1:90,2] + -0.052;
   1:L PR[91] R[100]mm/sec CNT100;
   1:  PR[GP1:91,1] = PR[GP1:90,1] + -67.402;
   1:  PR[GP1:91,2] = PR[GP1:90,2] + -1.190;
   1:L PR[91] R[100]mm/sec CNT100;
   1:  PR[GP1:91,1] = PR[GP1:90,1] + -66.898;
   1:  PR[GP1:91,2] = PR[GP1:90,2] + -6.883;
   1:L PR[91] R[100]mm/sec CNT100;
   1:  PR[GP1:91,1] = PR[GP1:90,1] + -65.236;
   1:  PR[GP1:91,2] = PR[GP1:90,2] + -12.529;
   1:L PR[91] R[100]mm/sec CNT100;
   1:  PR[GP1:91,1] = PR[GP1:90,1] + -62.075;
   1:  PR[GP1:91,2] = PR[GP1:90,2] + -18.778;
   1:L PR[91] R[100]mm/sec CNT100;
   1:  PR[GP1:91,1] = PR[GP1:90,1] + -58.047;
   1:  PR[GP1:91,2] = PR[GP1:90,2] + -24.021;
   1:L PR[91] R[100]mm/sec CNT100;
   1:  PR[GP1:91,1] = PR[GP1:90,1] + -53.509;
   1:  PR[GP1:91,2] = PR[GP1:90,2] + -28.090;
   1:L PR[91] R[100]mm/sec CNT100;
   1:  PR[GP1:91,1] = PR[GP1:90,1] + -52.545;
   1:  PR[GP1:91,2] = PR[GP1:90,2] + -28.868;
   1:L PR[91] R[100]mm/sec CNT100;
   1:  PR[GP1:91,1] = PR[GP1:90,1] + -47.314;
   1:  PR[GP1:91,2] = PR[GP1:90,2] + -32.127;
   1:L PR[91] R[100]mm/sec CNT100;
   1:  PR[GP1:91,1] = PR[GP1:90,1] + -42.204;
   1:  PR[GP1:91,2] = PR[GP1:90,2] + -34.179;
   1:L PR[91] R[100]mm/sec CNT100;
   1:  PR[GP1:91,1] = PR[GP1:90,1] + -39.546;
   1:  PR[GP1:91,2] = PR[GP1:90,2] + -35.116;
   1:L PR[91] R[100]mm/sec CNT100;
   1:  PR[GP1:91,1] = PR[GP1:90,1] + -34.294;
   1:  PR[GP1:91,2] = PR[GP1:90,2] + -36.249;
   1:L PR[91] R[100]mm/sec CNT100;
   1:  PR[GP1:91,1] = PR[GP1:90,1] + -29.538;
   1:  PR[GP1:91,2] = PR[GP1:90,2] + -36.433;
   1:L PR[91] R[100]mm/sec CNT100;
   1:  PR[GP1:91,1] = PR[GP1:90,1] + -25.102;
   1:  PR[GP1:91,2] = PR[GP1:90,2] + -36.447;
   1:L PR[91] R[100]mm/sec CNT100;
   1:  PR[GP1:91,1] = PR[GP1:90,1] + -20.608;
   1:  PR[GP1:91,2] = PR[GP1:90,2] + -35.859;
   1:L PR[91] R[100]mm/sec CNT100;
   1:  PR[GP1:91,1] = PR[GP1:90,1] + -16.762;
   1:  PR[GP1:91,2] = PR[GP1:90,2] + -34.636;
   1:L PR[91] R[100]mm/sec CNT100;
   1:  PR[GP1:91,1] = PR[GP1:90,1] + -11.297;
   1:  PR[GP1:91,2] = PR[GP1:90,2] + -32.737;
   1:L PR[91] R[100]mm/sec CNT100;
   1:  PR[GP1:91,1] = PR[GP1:90,1] + -7.968;
   1:  PR[GP1:91,2] = PR[GP1:90,2] + -30.995;
   1:L PR[91] R[100]mm/sec CNT100;
   1:  PR[GP1:91,1] = PR[GP1:90,1] + -4.321;
   1:  PR[GP1:91,2] = PR[GP1:90,2] + -28.345;
   1:L PR[91] R[100]mm/sec CNT100;
   1:  PR[GP1:91,1] = PR[GP1:90,1] + -3.761;
   1:  PR[GP1:91,2] = PR[GP1:90,2] + -27.906;
   1:L PR[91] R[100]mm/sec CNT100;
   1:  PR[GP1:91,1] = PR[GP1:90,1] + -3.227;
   1:  PR[GP1:91,2] = PR[GP1:90,2] + -27.287;
   1:L PR[91] R[100]mm/sec CNT100;
   1:  PR[GP1:91,1] = PR[GP1:90,1] + 0.536;
   1:  PR[GP1:91,2] = PR[GP1:90,2] + -26.479;
   1:L PR[91] R[100]mm/sec CNT100;
   1:  PR[GP1:91,1] = PR[GP1:90,1] + 1.134;
   1:  PR[GP1:91,2] = PR[GP1:90,2] + -26.162;
   1:L PR[91] R[100]mm/sec CNT100;
   1:  PR[GP1:91,1] = PR[GP1:90,1] + 3.492;
   1:  PR[GP1:91,2] = PR[GP1:90,2] + -27.351;
   1:L PR[91] R[100]mm/sec CNT100;
   1:  PR[GP1:91,1] = PR[GP1:90,1] + 3.976;
   1:  PR[GP1:91,2] = PR[GP1:90,2] + -27.914;
   1:L PR[91] R[100]mm/sec CNT100;
   1:  PR[GP1:91,1] = PR[GP1:90,1] + 4.534;
   1:  PR[GP1:91,2] = PR[GP1:90,2] + -28.350;
   1:L PR[91] R[100]mm/sec CNT100;
   1:  PR[GP1:91,1] = PR[GP1:90,1] + 8.189;
   1:  PR[GP1:91,2] = PR[GP1:90,2] + -31.005;
   1:L PR[91] R[100]mm/sec CNT100;
   1:  PR[GP1:91,1] = PR[GP1:90,1] + 11.491;
   1:  PR[GP1:91,2] = PR[GP1:90,2] + -32.728;
   1:L PR[91] R[100]mm/sec CNT100;
   1:  PR[GP1:91,1] = PR[GP1:90,1] + 15.589;
   1:  PR[GP1:91,2] = PR[GP1:90,2] + -34.045;
   1:L PR[91] R[100]mm/sec CNT100;
   1:  PR[GP1:91,1] = PR[GP1:90,1] + 20.824;
   1:  PR[GP1:91,2] = PR[GP1:90,2] + -35.857;
   1:L PR[91] R[100]mm/sec CNT100;
   1:  PR[GP1:91,1] = PR[GP1:90,1] + 25.294;
   1:  PR[GP1:91,2] = PR[GP1:90,2] + -36.445;
   1:L PR[91] R[100]mm/sec CNT100;
   1:  PR[GP1:91,1] = PR[GP1:90,1] + 30.515;
   1:  PR[GP1:91,2] = PR[GP1:90,2] + -36.270;
   1:L PR[91] R[100]mm/sec CNT100;
   1:  PR[GP1:91,1] = PR[GP1:90,1] + 34.484;
   1:  PR[GP1:91,2] = PR[GP1:90,2] + -36.252;
   1:L PR[91] R[100]mm/sec CNT100;
   1:  PR[GP1:91,1] = PR[GP1:90,1] + 39.707;
   1:  PR[GP1:91,2] = PR[GP1:90,2] + -35.128;
   1:L PR[91] R[100]mm/sec CNT100;
   1:  PR[GP1:91,1] = PR[GP1:90,1] + 45.438;
   1:  PR[GP1:91,2] = PR[GP1:90,2] + -32.870;
   1:L PR[91] R[100]mm/sec CNT100;
   1:  PR[GP1:91,1] = PR[GP1:90,1] + 47.508;
   1:  PR[GP1:91,2] = PR[GP1:90,2] + -32.137;
   1:L PR[91] R[100]mm/sec CNT100;
   1:  PR[GP1:91,1] = PR[GP1:90,1] + 52.683;
   1:  PR[GP1:91,2] = PR[GP1:90,2] + -28.929;
   1:L PR[91] R[100]mm/sec CNT100;
   1:  PR[GP1:91,1] = PR[GP1:90,1] + 57.707;
   1:  PR[GP1:91,2] = PR[GP1:90,2] + -24.480;
   1:L PR[91] R[100]mm/sec CNT100;
   1:  PR[GP1:91,1] = PR[GP1:90,1] + 58.188;
   1:  PR[GP1:91,2] = PR[GP1:90,2] + -24.091;
   1:L PR[91] R[100]mm/sec CNT100;
   1:  PR[GP1:91,1] = PR[GP1:90,1] + 62.248;
   1:  PR[GP1:91,2] = PR[GP1:90,2] + -18.820;
   1:L PR[91] R[100]mm/sec CNT100;
   1:  PR[GP1:91,1] = PR[GP1:90,1] + 65.423;
   1:  PR[GP1:91,2] = PR[GP1:90,2] + -12.615;
   1:L PR[91] R[100]mm/sec CNT100;
   1:  PR[GP1:91,1] = PR[GP1:90,1] + 67.092;
   1:  PR[GP1:91,2] = PR[GP1:90,2] + -7.025;
   1:L PR[91] R[100]mm/sec CNT100;
   1:  PR[GP1:91,1] = PR[GP1:90,1] + 67.254;
   1:  PR[GP1:91,2] = PR[GP1:90,2] + -5.983;
   1:L PR[91] R[100]mm/sec CNT100;
   1:  PR[GP1:91,1] = PR[GP1:90,1] + 67.795;
   1:  PR[GP1:91,2] = PR[GP1:90,2] + -0.092;
   1:L PR[91] R[100]mm/sec CNT100;
   1:  PR[GP1:91,1] = PR[GP1:90,1] + 67.615;
   1:  PR[GP1:91,2] = PR[GP1:90,2] + 1.049;
   1:L PR[91] R[100]mm/sec CNT100;
   1:  PR[GP1:91,1] = PR[GP1:90,1] + 67.086;
   1:  PR[GP1:91,2] = PR[GP1:90,2] + 6.900;
   1:L PR[91] R[100]mm/sec CNT100;
   1:  PR[GP1:91,1] = PR[GP1:90,1] + 65.423;
   1:  PR[GP1:91,2] = PR[GP1:90,2] + 12.471;
   1:L PR[91] R[100]mm/sec CNT100;
   1:  PR[GP1:91,1] = PR[GP1:90,1] + 62.278;
   1:  PR[GP1:91,2] = PR[GP1:90,2] + 18.625;
   1:L PR[91] R[100]mm/sec CNT100;
   1:  PR[GP1:91,1] = PR[GP1:90,1] + 58.179;
   1:  PR[GP1:91,2] = PR[GP1:90,2] + 23.959;
   1:L PR[91] R[100]mm/sec CNT100;
   1:  PR[GP1:91,1] = PR[GP1:90,1] + 53.666;
   1:  PR[GP1:91,2] = PR[GP1:90,2] + 27.994;
   1:L PR[91] R[100]mm/sec CNT100;
   1:  PR[GP1:91,1] = PR[GP1:90,1] + 52.696;
   1:  PR[GP1:91,2] = PR[GP1:90,2] + 28.777;
   1:L PR[91] R[100]mm/sec CNT100;
   1:  PR[GP1:91,1] = PR[GP1:90,1] + 47.499;
   1:  PR[GP1:91,2] = PR[GP1:90,2] + 31.998;
   1:L PR[91] R[100]mm/sec CNT100;
   1:  PR[GP1:91,1] = PR[GP1:90,1] + 42.383;
   1:  PR[GP1:91,2] = PR[GP1:90,2] + 34.042;
   1:L PR[91] R[100]mm/sec CNT100;
   1:  PR[GP1:91,1] = PR[GP1:90,1] + 39.721;
   1:  PR[GP1:91,2] = PR[GP1:90,2] + 34.981;
   1:L PR[91] R[100]mm/sec CNT100;
   1:  PR[GP1:91,1] = PR[GP1:90,1] + 34.479;
   1:  PR[GP1:91,2] = PR[GP1:90,2] + 36.110;
   1:L PR[91] R[100]mm/sec CNT100;
   1:  PR[GP1:91,1] = PR[GP1:90,1] + 29.747;
   1:  PR[GP1:91,2] = PR[GP1:90,2] + 36.288;
   1:L PR[91] R[100]mm/sec CNT100;
   1:  PR[GP1:91,1] = PR[GP1:90,1] + 25.311;
   1:  PR[GP1:91,2] = PR[GP1:90,2] + 36.304;
   1:L PR[91] R[100]mm/sec CNT100;
   1:  PR[GP1:91,1] = PR[GP1:90,1] + 20.824;
   1:  PR[GP1:91,2] = PR[GP1:90,2] + 35.714;
   1:L PR[91] R[100]mm/sec CNT100;
   1:  PR[GP1:91,1] = PR[GP1:90,1] + 16.974;
   1:  PR[GP1:91,2] = PR[GP1:90,2] + 34.489;
   1:L PR[91] R[100]mm/sec CNT100;
   1:  PR[GP1:91,1] = PR[GP1:90,1] + 11.506;
   1:  PR[GP1:91,2] = PR[GP1:90,2] + 32.593;
   1:L PR[91] R[100]mm/sec CNT100;
   1:  PR[GP1:91,1] = PR[GP1:90,1] + 8.191;
   1:  PR[GP1:91,2] = PR[GP1:90,2] + 30.863;
   1:L PR[91] R[100]mm/sec CNT100;
   1:  PR[GP1:91,1] = PR[GP1:90,1] + 5.542;
   1:  PR[GP1:91,2] = PR[GP1:90,2] + 28.991;
   1:L PR[91] R[100]mm/sec CNT100;
   1:  PR[GP1:91,1] = PR[GP1:90,1] + 4.412;
   1:  PR[GP1:91,2] = PR[GP1:90,2] + 28.108;
   1:L PR[91] R[100]mm/sec CNT100;
   1:  PR[GP1:91,1] = PR[GP1:90,1] + 3.476;
   1:  PR[GP1:91,2] = PR[GP1:90,2] + 27.018;
   1:L PR[91] R[100]mm/sec CNT100;
   1:  PR[GP1:91,1] = PR[GP1:90,1] + 1.802;
   1:  PR[GP1:91,2] = PR[GP1:90,2] + 26.357;
   1:L PR[91] R[100]mm/sec CNT100;
   1:  PR[GP1:91,1] = PR[GP1:90,1] + 1.249;
   1:  PR[GP1:91,2] = PR[GP1:90,2] + 26.074;
   1:L PR[91] R[100]mm/sec CNT100;
   1:  ! -- Layer/Ebene 88 -- !;
   1:  PR[91] = PR[90];
   1:  PR[GP1:91,1] = PR[GP1:90,1] + -2.365;
   1:  PR[GP1:91,2] = PR[GP1:90,2] + 26.874;
   1:  PR[GP1:91,3] = PR[GP1:90,3] + 53.985;
   1:L PR[91] R[100]mm/sec CNT100;
   1:  PR[GP1:91,1] = PR[GP1:90,1] + -3.255;
   1:  PR[GP1:91,2] = PR[GP1:90,2] + 27.327;
   1:L PR[91] R[100]mm/sec CNT100;
   1:  PR[GP1:91,1] = PR[GP1:90,1] + -4.037;
   1:  PR[GP1:91,2] = PR[GP1:90,2] + 28.236;
   1:L PR[91] R[100]mm/sec CNT100;
   1:  PR[GP1:91,1] = PR[GP1:90,1] + -4.998;
   1:  PR[GP1:91,2] = PR[GP1:90,2] + 28.989;
   1:L PR[91] R[100]mm/sec CNT100;
   1:  PR[GP1:91,1] = PR[GP1:90,1] + -7.760;
   1:  PR[GP1:91,2] = PR[GP1:90,2] + 30.940;
   1:L PR[91] R[100]mm/sec CNT100;
   1:  PR[GP1:91,1] = PR[GP1:90,1] + -10.958;
   1:  PR[GP1:91,2] = PR[GP1:90,2] + 32.613;
   1:L PR[91] R[100]mm/sec CNT100;
   1:  PR[GP1:91,1] = PR[GP1:90,1] + -14.895;
   1:  PR[GP1:91,2] = PR[GP1:90,2] + 33.878;
   1:L PR[91] R[100]mm/sec CNT100;
   1:  PR[GP1:91,1] = PR[GP1:90,1] + -20.425;
   1:  PR[GP1:91,2] = PR[GP1:90,2] + 35.790;
   1:L PR[91] R[100]mm/sec CNT100;
   1:  PR[GP1:91,1] = PR[GP1:90,1] + -24.748;
   1:  PR[GP1:91,2] = PR[GP1:90,2] + 36.355;
   1:L PR[91] R[100]mm/sec CNT100;
   1:  PR[GP1:91,1] = PR[GP1:90,1] + -29.817;
   1:  PR[GP1:91,2] = PR[GP1:90,2] + 36.181;
   1:L PR[91] R[100]mm/sec CNT100;
   1:  PR[GP1:91,1] = PR[GP1:90,1] + -34.120;
   1:  PR[GP1:91,2] = PR[GP1:90,2] + 36.159;
   1:L PR[91] R[100]mm/sec CNT100;
   1:  PR[GP1:91,1] = PR[GP1:90,1] + -39.193;
   1:  PR[GP1:91,2] = PR[GP1:90,2] + 35.065;
   1:L PR[91] R[100]mm/sec CNT100;
   1:  PR[GP1:91,1] = PR[GP1:90,1] + -44.746;
   1:  PR[GP1:91,2] = PR[GP1:90,2] + 32.866;
   1:L PR[91] R[100]mm/sec CNT100;
   1:  PR[GP1:91,1] = PR[GP1:90,1] + -47.142;
   1:  PR[GP1:91,2] = PR[GP1:90,2] + 32.015;
   1:L PR[91] R[100]mm/sec CNT100;
   1:  PR[GP1:91,1] = PR[GP1:90,1] + -52.209;
   1:  PR[GP1:91,2] = PR[GP1:90,2] + 28.859;
   1:L PR[91] R[100]mm/sec CNT100;
   1:  PR[GP1:91,1] = PR[GP1:90,1] + -57.125;
   1:  PR[GP1:91,2] = PR[GP1:90,2] + 24.494;
   1:L PR[91] R[100]mm/sec CNT100;
   1:  PR[GP1:91,1] = PR[GP1:90,1] + -57.873;
   1:  PR[GP1:91,2] = PR[GP1:90,2] + 23.889;
   1:L PR[91] R[100]mm/sec CNT100;
   1:  PR[GP1:91,1] = PR[GP1:90,1] + -61.791;
   1:  PR[GP1:91,2] = PR[GP1:90,2] + 18.788;
   1:L PR[91] R[100]mm/sec CNT100;
   1:  PR[GP1:91,1] = PR[GP1:90,1] + -65.020;
   1:  PR[GP1:91,2] = PR[GP1:90,2] + 12.509;
   1:L PR[91] R[100]mm/sec CNT100;
   1:  PR[GP1:91,1] = PR[GP1:90,1] + -66.787;
   1:  PR[GP1:91,2] = PR[GP1:90,2] + 6.506;
   1:L PR[91] R[100]mm/sec CNT100;
   1:  PR[GP1:91,1] = PR[GP1:90,1] + -66.860;
   1:  PR[GP1:91,2] = PR[GP1:90,2] + 6.038;
   1:L PR[91] R[100]mm/sec CNT100;
   1:  PR[GP1:91,1] = PR[GP1:90,1] + -67.407;
   1:  PR[GP1:91,2] = PR[GP1:90,2] + -0.052;
   1:L PR[91] R[100]mm/sec CNT100;
   1:  PR[GP1:91,1] = PR[GP1:90,1] + -67.315;
   1:  PR[GP1:91,2] = PR[GP1:90,2] + -0.637;
   1:L PR[91] R[100]mm/sec CNT100;
   1:  PR[GP1:91,1] = PR[GP1:90,1] + -66.782;
   1:  PR[GP1:91,2] = PR[GP1:90,2] + -6.669;
   1:L PR[91] R[100]mm/sec CNT100;
   1:  PR[GP1:91,1] = PR[GP1:90,1] + -65.019;
   1:  PR[GP1:91,2] = PR[GP1:90,2] + -12.655;
   1:L PR[91] R[100]mm/sec CNT100;
   1:  PR[GP1:91,1] = PR[GP1:90,1] + -61.975;
   1:  PR[GP1:91,2] = PR[GP1:90,2] + -18.631;
   1:L PR[91] R[100]mm/sec CNT100;
   1:  PR[GP1:91,1] = PR[GP1:90,1] + -61.803;
   1:  PR[GP1:91,2] = PR[GP1:90,2] + -18.916;
   1:L PR[91] R[100]mm/sec CNT100;
   1:  PR[GP1:91,1] = PR[GP1:90,1] + -57.863;
   1:  PR[GP1:91,2] = PR[GP1:90,2] + -24.045;
   1:L PR[91] R[100]mm/sec CNT100;
   1:  PR[GP1:91,1] = PR[GP1:90,1] + -53.439;
   1:  PR[GP1:91,2] = PR[GP1:90,2] + -28.013;
   1:L PR[91] R[100]mm/sec CNT100;
   1:  PR[GP1:91,1] = PR[GP1:90,1] + -52.219;
   1:  PR[GP1:91,2] = PR[GP1:90,2] + -28.996;
   1:L PR[91] R[100]mm/sec CNT100;
   1:  PR[GP1:91,1] = PR[GP1:90,1] + -47.130;
   1:  PR[GP1:91,2] = PR[GP1:90,2] + -32.167;
   1:L PR[91] R[100]mm/sec CNT100;
   1:  PR[GP1:91,1] = PR[GP1:90,1] + -42.158;
   1:  PR[GP1:91,2] = PR[GP1:90,2] + -34.163;
   1:L PR[91] R[100]mm/sec CNT100;
   1:  PR[GP1:91,1] = PR[GP1:90,1] + -39.200;
   1:  PR[GP1:91,2] = PR[GP1:90,2] + -35.207;
   1:L PR[91] R[100]mm/sec CNT100;
   1:  PR[GP1:91,1] = PR[GP1:90,1] + -34.106;
   1:  PR[GP1:91,2] = PR[GP1:90,2] + -36.306;
   1:L PR[91] R[100]mm/sec CNT100;
   1:  PR[GP1:91,1] = PR[GP1:90,1] + -29.493;
   1:  PR[GP1:91,2] = PR[GP1:90,2] + -36.484;
   1:L PR[91] R[100]mm/sec CNT100;
   1:  PR[GP1:91,1] = PR[GP1:90,1] + -24.749;
   1:  PR[GP1:91,2] = PR[GP1:90,2] + -36.499;
   1:L PR[91] R[100]mm/sec CNT100;
   1:  PR[GP1:91,1] = PR[GP1:90,1] + -20.409;
   1:  PR[GP1:91,2] = PR[GP1:90,2] + -35.931;
   1:L PR[91] R[100]mm/sec CNT100;
   1:  PR[GP1:91,1] = PR[GP1:90,1] + -16.693;
   1:  PR[GP1:91,2] = PR[GP1:90,2] + -34.749;
   1:L PR[91] R[100]mm/sec CNT100;
   1:  PR[GP1:91,1] = PR[GP1:90,1] + -10.955;
   1:  PR[GP1:91,2] = PR[GP1:90,2] + -32.755;
   1:L PR[91] R[100]mm/sec CNT100;
   1:  PR[GP1:91,1] = PR[GP1:90,1] + -7.757;
   1:  PR[GP1:91,2] = PR[GP1:90,2] + -31.082;
   1:L PR[91] R[100]mm/sec CNT100;
   1:  PR[GP1:91,1] = PR[GP1:90,1] + -3.947;
   1:  PR[GP1:91,2] = PR[GP1:90,2] + -28.314;
   1:L PR[91] R[100]mm/sec CNT100;
   1:  PR[GP1:91,1] = PR[GP1:90,1] + -3.588;
   1:  PR[GP1:91,2] = PR[GP1:90,2] + -28.032;
   1:L PR[91] R[100]mm/sec CNT100;
   1:  PR[GP1:91,1] = PR[GP1:90,1] + -3.198;
   1:  PR[GP1:91,2] = PR[GP1:90,2] + -27.580;
   1:L PR[91] R[100]mm/sec CNT100;
   1:  PR[GP1:91,1] = PR[GP1:90,1] + 0.703;
   1:  PR[GP1:91,2] = PR[GP1:90,2] + -26.743;
   1:L PR[91] R[100]mm/sec CNT100;
   1:  PR[GP1:91,1] = PR[GP1:90,1] + 1.175;
   1:  PR[GP1:91,2] = PR[GP1:90,2] + -26.492;
   1:L PR[91] R[100]mm/sec CNT100;
   1:  PR[GP1:91,1] = PR[GP1:90,1] + 3.462;
   1:  PR[GP1:91,2] = PR[GP1:90,2] + -27.644;
   1:L PR[91] R[100]mm/sec CNT100;
   1:  PR[GP1:91,1] = PR[GP1:90,1] + 3.801;
   1:  PR[GP1:91,2] = PR[GP1:90,2] + -28.038;
   1:L PR[91] R[100]mm/sec CNT100;
   1:  PR[GP1:91,1] = PR[GP1:90,1] + 4.159;
   1:  PR[GP1:91,2] = PR[GP1:90,2] + -28.318;
   1:L PR[91] R[100]mm/sec CNT100;
   1:  PR[GP1:91,1] = PR[GP1:90,1] + 7.977;
   1:  PR[GP1:91,2] = PR[GP1:90,2] + -31.092;
   1:L PR[91] R[100]mm/sec CNT100;
   1:  PR[GP1:91,1] = PR[GP1:90,1] + 11.149;
   1:  PR[GP1:91,2] = PR[GP1:90,2] + -32.747;
   1:L PR[91] R[100]mm/sec CNT100;
   1:  PR[GP1:91,1] = PR[GP1:90,1] + 15.088;
   1:  PR[GP1:91,2] = PR[GP1:90,2] + -34.012;
   1:L PR[91] R[100]mm/sec CNT100;
   1:  PR[GP1:91,1] = PR[GP1:90,1] + 20.625;
   1:  PR[GP1:91,2] = PR[GP1:90,2] + -35.930;
   1:L PR[91] R[100]mm/sec CNT100;
   1:  PR[GP1:91,1] = PR[GP1:90,1] + 24.942;
   1:  PR[GP1:91,2] = PR[GP1:90,2] + -36.497;
   1:L PR[91] R[100]mm/sec CNT100;
   1:  PR[GP1:91,1] = PR[GP1:90,1] + 29.987;
   1:  PR[GP1:91,2] = PR[GP1:90,2] + -36.328;
   1:L PR[91] R[100]mm/sec CNT100;
   1:  PR[GP1:91,1] = PR[GP1:90,1] + 34.297;
   1:  PR[GP1:91,2] = PR[GP1:90,2] + -36.309;
   1:L PR[91] R[100]mm/sec CNT100;
   1:  PR[GP1:91,1] = PR[GP1:90,1] + 39.362;
   1:  PR[GP1:91,2] = PR[GP1:90,2] + -35.219;
   1:L PR[91] R[100]mm/sec CNT100;
   1:  PR[GP1:91,1] = PR[GP1:90,1] + 44.923;
   1:  PR[GP1:91,2] = PR[GP1:90,2] + -33.028;
   1:L PR[91] R[100]mm/sec CNT100;
   1:  PR[GP1:91,1] = PR[GP1:90,1] + 47.325;
   1:  PR[GP1:91,2] = PR[GP1:90,2] + -32.177;
   1:L PR[91] R[100]mm/sec CNT100;
   1:  PR[GP1:91,1] = PR[GP1:90,1] + 52.360;
   1:  PR[GP1:91,2] = PR[GP1:90,2] + -29.056;
   1:L PR[91] R[100]mm/sec CNT100;
   1:  PR[GP1:91,1] = PR[GP1:90,1] + 57.249;
   1:  PR[GP1:91,2] = PR[GP1:90,2] + -24.726;
   1:L PR[91] R[100]mm/sec CNT100;
   1:  PR[GP1:91,1] = PR[GP1:90,1] + 58.006;
   1:  PR[GP1:91,2] = PR[GP1:90,2] + -24.113;
   1:L PR[91] R[100]mm/sec CNT100;
   1:  PR[GP1:91,1] = PR[GP1:90,1] + 61.965;
   1:  PR[GP1:91,2] = PR[GP1:90,2] + -18.973;
   1:L PR[91] R[100]mm/sec CNT100;
   1:  PR[GP1:91,1] = PR[GP1:90,1] + 65.206;
   1:  PR[GP1:91,2] = PR[GP1:90,2] + -12.743;
   1:L PR[91] R[100]mm/sec CNT100;
   1:  PR[GP1:91,1] = PR[GP1:90,1] + 66.974;
   1:  PR[GP1:91,2] = PR[GP1:90,2] + -6.819;
   1:L PR[91] R[100]mm/sec CNT100;
   1:  PR[GP1:91,1] = PR[GP1:90,1] + 67.045;
   1:  PR[GP1:91,2] = PR[GP1:90,2] + -6.357;
   1:L PR[91] R[100]mm/sec CNT100;
   1:  PR[GP1:91,1] = PR[GP1:90,1] + 67.621;
   1:  PR[GP1:91,2] = PR[GP1:90,2] + -0.092;
   1:L PR[91] R[100]mm/sec CNT100;
   1:  PR[GP1:91,1] = PR[GP1:90,1] + 67.528;
   1:  PR[GP1:91,2] = PR[GP1:90,2] + 0.494;
   1:L PR[91] R[100]mm/sec CNT100;
   1:  PR[GP1:91,1] = PR[GP1:90,1] + 66.968;
   1:  PR[GP1:91,2] = PR[GP1:90,2] + 6.693;
   1:L PR[91] R[100]mm/sec CNT100;
   1:  PR[GP1:91,1] = PR[GP1:90,1] + 65.205;
   1:  PR[GP1:91,2] = PR[GP1:90,2] + 12.600;
   1:L PR[91] R[100]mm/sec CNT100;
   1:  PR[GP1:91,1] = PR[GP1:90,1] + 62.151;
   1:  PR[GP1:91,2] = PR[GP1:90,2] + 18.525;
   1:L PR[91] R[100]mm/sec CNT100;
   1:  PR[GP1:91,1] = PR[GP1:90,1] + 61.977;
   1:  PR[GP1:91,2] = PR[GP1:90,2] + 18.814;
   1:L PR[91] R[100]mm/sec CNT100;
